   //........................Присваиваем обработанный выход к физическим выходам модуля...............................................................

   "AO V11.1" := "__MainBlock".Valve_Regul[1].iAnalogOutput;

   "AO V12.1" := "__MainBlock".Valve_Regul[2].iAnalogOutput;

   "AO V3 (NO)" := "__MainBlock".Valve_Regul[3].iAnalogOutput;

   //========================  Управление выходом пневмоострова для клапана регулировки============================
   //Управление клапанами через тройник от выходов запорных клапанов V11 и V12
   "__MainBlock".Valve_Regul[1].bAutoOpenClose := "V11_Запорный тепло";  //Сигнал на открытие регулировочного клапана паралельно с запорным клапаном
   "__MainBlock".Valve_Regul[2].bAutoOpenClose := "V12_Запор гликоль" ;   //Сигнал на открытие регулировочного клапана паралельно с запорным клапаном

   // Выход для управления клапаном V3
   "V3_Давления" := "__MainBlock".Valve_Regul[3].bOut_OpenClose;

   //=======================================//=======================================//=======================================//=======================================

   "__MainBlock".Valve_Regul[1].bManualOpenClose := "__MainBlock"."Valve_o/c"[11].bManualOpen;

   "__MainBlock".Valve_Regul[2].bManualOpenClose := "__MainBlock"."Valve_o/c"[12].bManualOpen;
END_FUNCTION

FUNCTION "Расчет ПЕ1" : Void   // FC9, LAD
{ S7_Optimized_Access := 'FALSE' }
VERSION : 0.1
   VAR_INPUT
      "ПЕ (ед)" : Int;
      "Выдержка (сек)" : Int;
      "Производит установки (л\ч)" : Int;
      "Производит заданная (л\ч)" : Int;
      "Уст.Темп (С)" : Real;   // Уставка температуры нагрева продукта
      "Выбор уставки для температуры (0 - ПЕ, 1 - Те)" : Bool;   // Для выбора от куда брать уставку температуры или вводим ПЕ и расчитываем ТЕ или просто вводим желаемую ПЕ
   END_VAR
   VAR_OUTPUT
      "Температура пастеризации" : Real;   // уставка для ПИД нагрева. Или расчитываем по ПЕ или по уставке желаемой ТЕ
      "Выдержка реальная_1" : Int;
      "Расчтеная ПЕ по Те" : Real;   // Расчет ПЕ по уставке Те для HMI
   END_VAR
   VAR_TEMP
      "1" : Real;
      "выдержка реальная" : Int;
      "2" : UInt;
      "3" : Real;
      "4" : Real;
      "5" : Real;
      "6" : Real;
      "Расчетная темп по ПЕ" : Real;   // Расчет температуры по уставке ПЕ
      "PE/10" : Int;
   END_VAR
   VAR CONSTANT
      "1.393" : Real := 1.393;
      "60" : Real := 60.0;
   END_VAR
BEGIN

REGION Network 1
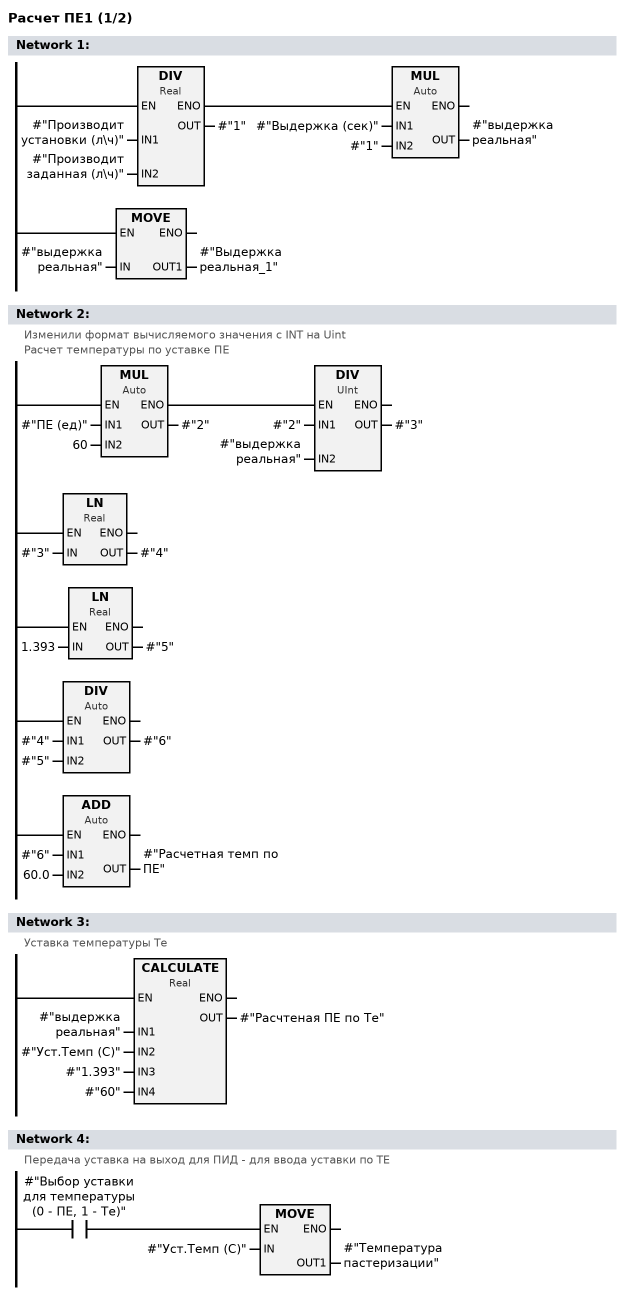
   RUNG wire#powerrail
      { S7_Templates := "SrcType := Real" } Div(in1 := #"Производит установки (л\ч)", in2 := #"Производит заданная (л\ч)", out => #"1")
      Mul(in1 := #"Выдержка (сек)", in2 := #"1", out => #"выдержка реальная")
   END_RUNG
   RUNG wire#powerrail
      Move(in := #"выдержка реальная", out1 => #"Выдержка реальная_1")
   END_RUNG
   // the same network as SCL:
   #"1" := #"Производит установки (л\ч)" / #"Производит заданная (л\ч)";
   #"выдержка реальная" := #"Выдержка (сек)" * #"1";
   #"Выдержка реальная_1" := #"выдержка реальная";
END_REGION

REGION Network 2
   // Изменили формат вычисляемого значения с INT на Uint
   // Расчет температуры по уставке ПЕ
   #"2" := #"ПЕ (ед)" * 60;
   #"3" := #"2" / #"выдержка реальная";
   #"4" := LN(#"3");
   #"5" := LN(1.393);
   #"6" := #"4" / #"5";
   #"Расчетная темп по ПЕ" := #"6" + 60.0;
END_REGION

REGION Network 3
   // Уставка температуры Те
   RUNG wire#powerrail
      { S7_Templates := "SrcType := Real"; S7_Expression := "IN1/IN4*(IN3**(IN2-IN4))" } Calculate(in1 := #"выдержка реальная", in2 := #"Уст.Темп (С)", in3 := #"1.393", in4 := #"60", out => #"Расчтеная ПЕ по Те")
   END_RUNG
   // the same network as SCL:
   #"Расчтеная ПЕ по Те" := #"выдержка реальная"/#"60"*(#"1.393"**(#"Уст.Темп (С)"-#"60"));
END_REGION

REGION Network 4
   // Передача уставка на выход для ПИД - для ввода уставки по ТЕ
   RUNG wire#powerrail
      Contact( #"Выбор уставки для температуры (0 - ПЕ, 1 - Те)" )
      Move(in := #"Уст.Темп (С)", out1 => #"Температура пастеризации")
   END_RUNG
   // the same network as SCL:
   IF #"Выбор уставки для температуры (0 - ПЕ, 1 - Те)" THEN
       #"Температура пастеризации" := #"Уст.Темп (С)";
   END_IF;
END_REGION

REGION Network 5
   // Передача уставка на выход для ПИД - для ввода уставки по ПЕ
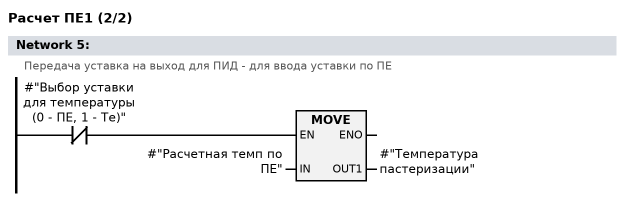
   RUNG wire#powerrail
      I_Contact( #"Выбор уставки для температуры (0 - ПЕ, 1 - Те)" )
      Move(in := #"Расчетная темп по ПЕ", out1 => #"Температура пастеризации")
   END_RUNG
   // the same network as SCL:
   IF NOT #"Выбор уставки для температуры (0 - ПЕ, 1 - Те)" THEN
       #"Температура пастеризации" := #"Расчетная темп по ПЕ";
   END_IF;
END_REGION
END_FUNCTION

FUNCTION "Все в Авто" : Void   // FC12, SCL
{ S7_Optimized_Access := 'TRUE' }
VERSION : 0.1
   VAR_TEMP
      fTrig_All_Auto : Bool;   // Фронт нажития кнопки все в авто
      i : Int;
   END_VAR
BEGIN

   //Отлавливаем фронт нажатия клавиши все в авто
   "R_trig_All_Auto"(In:="Клапана  в автомат",
                     Q=>#fTrig_All_Auto);

   //Сбрасываем все ручное в автоматический режим
   //
   IF #fTrig_All_Auto THEN

       //симуляция датчиков аналоговых
       //
       FOR #i := 1 TO 12 DO
           "__MainBlock".AI[#i].bSimEnable := FALSE;
       END_FOR;


       //Управление Valve o/c 
       FOR #i := 1 TO 20 DO
           "__MainBlock"."Valve_o/c"[#i].bManualMode := FALSE;
       END_FOR;

       //Управление Valve regul 
       FOR #i := 1 TO 3 DO
           "__MainBlock".Valve_Regul[#i].bManualMode := FALSE;
       END_FOR;


       //Управление Pumps
       FOR #i := 1 TO 6 DO
           "__MainBlock".Pump[#i].bManualMode := FALSE;
       END_FOR;



       //DI
       (*
       "DI".DI_0.bSimulation := FALSE;
       "DI".DI_1.bSimulation := FALSE;
       "DI".DI_2.bSimulation := FALSE;
       "DI".DI_3.bSimulation := FALSE;
       "DI".DI_4.bSimulation := FALSE;
       "DI".DI_5.bSimulation := FALSE;
       "DI".DI_6.bSimulation := FALSE;
       "DI".DI_7.bSimulation := FALSE;
       "DI".DI_8.bSimulation := FALSE;
       "DI".DI_9.bSimulation := FALSE;
       "DI".DI_10.bSimulation := FALSE;
       "DI".DI_11.bSimulation := FALSE;
       "DI".DI_12.bSimulation := FALSE;
       "DI".DI_13.bSimulation := FALSE;
       "DI".DI_14.bSimulation := FALSE;
       "DI".DI_15.bSimulation := FALSE;
       "DI".DI_16.bSimulation := FALSE;
       "DI".DI_17.bSimulation := FALSE;
       "DI".DI_18.bSimulation := FALSE;
       "DI".DI_19.bSimulation := FALSE;
       "DI".DI_20.bSimulation := FALSE;
       "DI".DI_21.bSimulation := FALSE;
       "DI".DI_22.bSimulation := FALSE;
       "DI".DI_23.bSimulation := FALSE;
       "DI".DI_24.bSimulation := FALSE;
       "DI".DI_25.bSimulation := FALSE;
       "DI".DI_26.bSimulation := FALSE;
       "DI".DI_27.bSimulation := FALSE;
       "DI".DI_28.bSimulation := FALSE;
       "DI".DI_29.bSimulation := FALSE;
      *)
   END_IF;
END_FUNCTION

FUNCTION "RestetAlarms" : Void   // FC13, SCL
{ S7_Optimized_Access := 'TRUE' }
VERSION : 0.1
   VAR_TEMP
      i : Int;
   END_VAR
BEGIN
   IF "bHMI_ResetAlarm" THEN

       //Сброс аварий насосов
       //
       FOR #i := 1 TO 6 DO
           "__MainBlock".Pump[#i].bResAlarm := TRUE;
       END_FOR;

       //Сброс аварий клапана
       //
       FOR #i := 1 TO 20 DO
           "__MainBlock"."Valve_o/c"[#i].bResetAlarm := TRUE;
       END_FOR;

   ELSE

       //Сброс аварий клапана
       FOR #i := 1 TO 20 DO
           "__MainBlock"."Valve_o/c"[#i].bResetAlarm := FALSE;
       END_FOR;

       //Сброс аварий насосов
       //
       FOR #i := 1 TO 6 DO
           "__MainBlock".Pump[#i].bResAlarm := FALSE;
       END_FOR;

   END_IF;
END_FUNCTION

ORGANIZATION_BLOCK "Main"   // OB1, LAD, ProgramCycle
TITLE = "Main Program Sweep (Cycle)"
{ S7_Optimized_Access := 'TRUE' }
AUTHOR : Алексей
VERSION : 0.1
   VAR_INPUT
      Initial_Call : Bool;   // Initial call of this OB
      Remanence : Bool;   // =True, if remanent data are available
   END_VAR
BEGIN

REGION Network 1: Расчет ПЕ
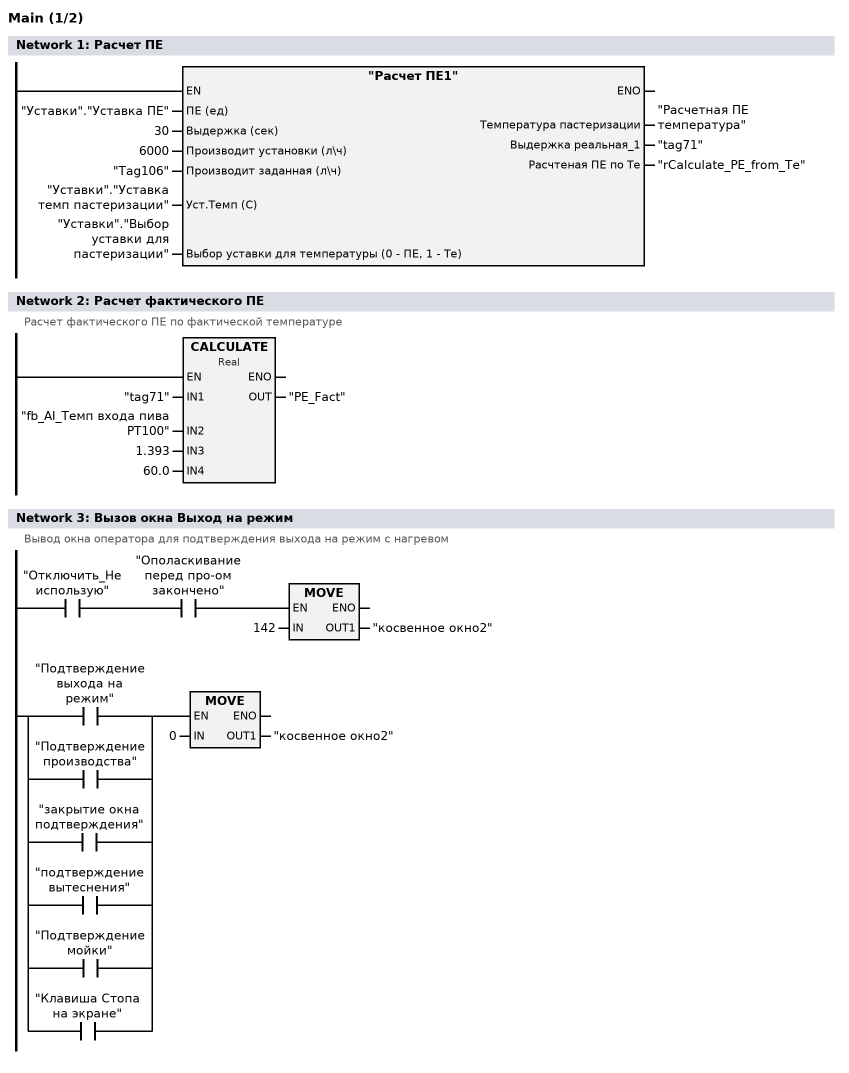
   RUNG wire#powerrail
      "Расчет ПЕ1"("ПЕ (ед)" := "Уставки"."Уставка ПЕ", "Выдержка (сек)" := 30, "Производит установки (л\ч)" := 6000, "Производит заданная (л\ч)" := "Tag106", "Уст.Темп (С)" := "Уставки"."Уставка темп пастеризации", "Выбор уставки для температуры (0 - ПЕ, 1 - Те)" := "Уставки"."Выбор уставки для пастеризации", "Температура пастеризации" => "Расчетная ПЕ температура", "Выдержка реальная_1" => "tag71", "Расчтеная ПЕ по Те" => "rCalculate_PE_from_Te")
   END_RUNG
   // the same network as SCL:
   "Расчет ПЕ1"("ПЕ (ед)" := "Уставки"."Уставка ПЕ",
                "Выдержка (сек)" := 30,
                "Производит установки (л\ч)" := 6000,
                "Производит заданная (л\ч)" := "Tag106",
                "Уст.Темп (С)" := "Уставки"."Уставка темп пастеризации",
                "Выбор уставки для температуры (0 - ПЕ, 1 - Те)" := "Уставки"."Выбор уставки для пастеризации",
                "Температура пастеризации" => "Расчетная ПЕ температура",
                "Выдержка реальная_1" => "tag71",
                "Расчтеная ПЕ по Те" => "rCalculate_PE_from_Te");
END_REGION

REGION Network 2: Расчет фактического ПЕ
   // Расчет фактического ПЕ по фактической температуре
   RUNG wire#powerrail
      { S7_Templates := "SrcType := Real"; S7_Expression := "IN1/IN4*(IN3**(IN2-IN4))" } Calculate(in1 := "tag71", in2 := "fb_AI_Темп входа пива PT100", in3 := 1.393, in4 := 60.0, out => "PE_Fact")
   END_RUNG
   // the same network as SCL:
   "PE_Fact" := "tag71"/60.0*(1.393**("fb_AI_Темп входа пива PT100"-60.0));
END_REGION

REGION Network 3: Вызов окна Выход на режим
   // Вывод окна оператора для подтверждения выхода на режим с нагревом
   RUNG wire#powerrail
      Contact( "Отключить_Не использую" )
      Contact( "Ополаскивание перед про-ом закончено" )
      Move(in := 142, out1 => "косвенное окно2")
   END_RUNG
   RUNG wire#powerrail
      Contact( "Подтверждение выхода на режим" )
      wire#w1
      Move(in := 0, out1 => "косвенное окно2")
   END_RUNG
   RUNG wire#powerrail
      Contact( "Подтверждение производства" )
   END_RUNG wire#w1
   RUNG wire#powerrail
      Contact( "закрытие окна подтверждения" )
   END_RUNG wire#w1
   RUNG wire#powerrail
      Contact( "подтверждение вытеснения" )
   END_RUNG wire#w1
   RUNG wire#powerrail
      Contact( "Подтверждение мойки" )
   END_RUNG wire#w1
   RUNG wire#powerrail
      Contact( "Клавиша Стопа на экране" )
   END_RUNG wire#w1
   // the same network as SCL:
   IF "Отключить_Не использую" AND "Ополаскивание перед про-ом закончено" THEN
       "косвенное окно2" := 142;
   END_IF;
   IF "Подтверждение выхода на режим" OR "Подтверждение производства" OR "закрытие окна подтверждения" OR "подтверждение вытеснения" OR "Подтверждение мойки" OR "Клавиша Стопа на экране" THEN
       "косвенное окно2" := 0;
   END_IF;
END_REGION

REGION Network 4: 11
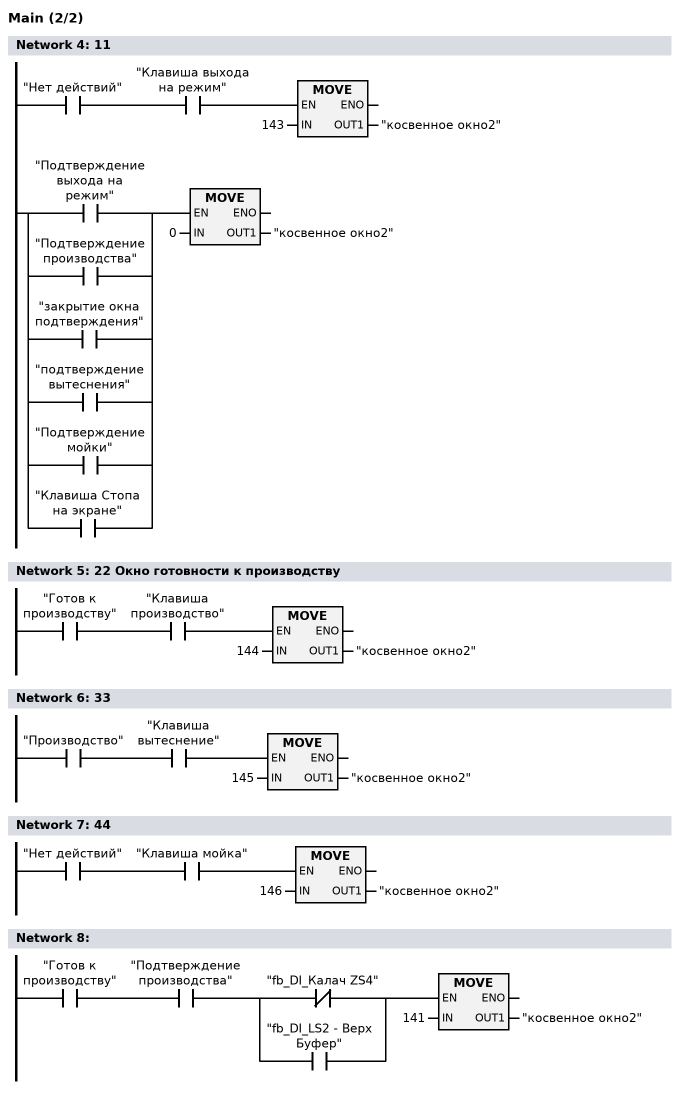
   RUNG wire#powerrail
      Contact( "Нет действий" )
      Contact( "Клавиша выхода на режим" )
      Move(in := 143, out1 => "косвенное окно2")
   END_RUNG
   RUNG wire#powerrail
      Contact( "Подтверждение выхода на режим" )
      wire#w1
      Move(in := 0, out1 => "косвенное окно2")
   END_RUNG
   RUNG wire#powerrail
      Contact( "Подтверждение производства" )
   END_RUNG wire#w1
   RUNG wire#powerrail
      Contact( "закрытие окна подтверждения" )
   END_RUNG wire#w1
   RUNG wire#powerrail
      Contact( "подтверждение вытеснения" )
   END_RUNG wire#w1
   RUNG wire#powerrail
      Contact( "Подтверждение мойки" )
   END_RUNG wire#w1
   RUNG wire#powerrail
      Contact( "Клавиша Стопа на экране" )
   END_RUNG wire#w1
   // the same network as SCL:
   IF "Нет действий" AND "Клавиша выхода на режим" THEN "косвенное окно2" := 143; END_IF;
   IF "Подтверждение выхода на режим" OR "Подтверждение производства" OR "закрытие окна подтверждения" OR "подтверждение вытеснения" OR "Подтверждение мойки" OR "Клавиша Стопа на экране" THEN
       "косвенное окно2" := 0;
   END_IF;
END_REGION

REGION Network 5: 22 Окно готовности к производству
   RUNG wire#powerrail
      Contact( "Готов к производству" )
      Contact( "Клавиша производство" )
      Move(in := 144, out1 => "косвенное окно2")
   END_RUNG
   // the same network as SCL:
   IF "Готов к производству" AND "Клавиша производство" THEN "косвенное окно2" := 144; END_IF;
END_REGION

REGION Network 6: 33
   RUNG wire#powerrail
      Contact( "Производство" )
      Contact( "Клавиша вытеснение" )
      Move(in := 145, out1 => "косвенное окно2")
   END_RUNG
   // the same network as SCL:
   IF "Производство" AND "Клавиша вытеснение" THEN "косвенное окно2" := 145; END_IF;
END_REGION

REGION Network 7: 44
   RUNG wire#powerrail
      Contact( "Нет действий" )
      Contact( "Клавиша мойка" )
      Move(in := 146, out1 => "косвенное окно2")
   END_RUNG
   // the same network as SCL:
   IF "Нет действий" AND "Клавиша мойка" THEN "косвенное окно2" := 146; END_IF;
END_REGION

REGION Network 8
   RUNG wire#powerrail
      Contact( "Готов к производству" )
      Contact( "Подтверждение производства" )
      wire#w1
      I_Contact( "fb_DI_Калач ZS4" )
      wire#w2
      Move(in := 141, out1 => "косвенное окно2")
   END_RUNG
   RUNG wire#w1
      Contact( "fb_DI_LS2 - Верх Буфер" )
   END_RUNG wire#w2
   // the same network as SCL:
   IF "Готов к производству" AND "Подтверждение производства" AND (NOT "fb_DI_Калач ZS4" OR "fb_DI_LS2 - Верх Буфер") THEN
       "косвенное окно2" := 141;
   END_IF;
END_REGION
END_ORGANIZATION_BLOCK

ORGANIZATION_BLOCK "Масштабирование"   // OB123, LAD, ProgramCycle
TITLE = "Main Program Sweep (Cycle)"
{ S7_Optimized_Access := 'TRUE' }
VERSION : 0.1
   VAR_INPUT
      Initial_Call : Bool;   // Initial call of this OB
      Remanence : Bool;   // =True, if remanent data are available
   END_VAR
   VAR_TEMP
      a1 : Real;
      a2 : Real;
      a3 : Real;
      a4 : Real;
      a5 : Real;
      a6 : Real;
      a7 : Real;
      a8 : Real;
      a9 : Real;
   END_VAR
BEGIN

REGION Network 1: Температура выхода продукта
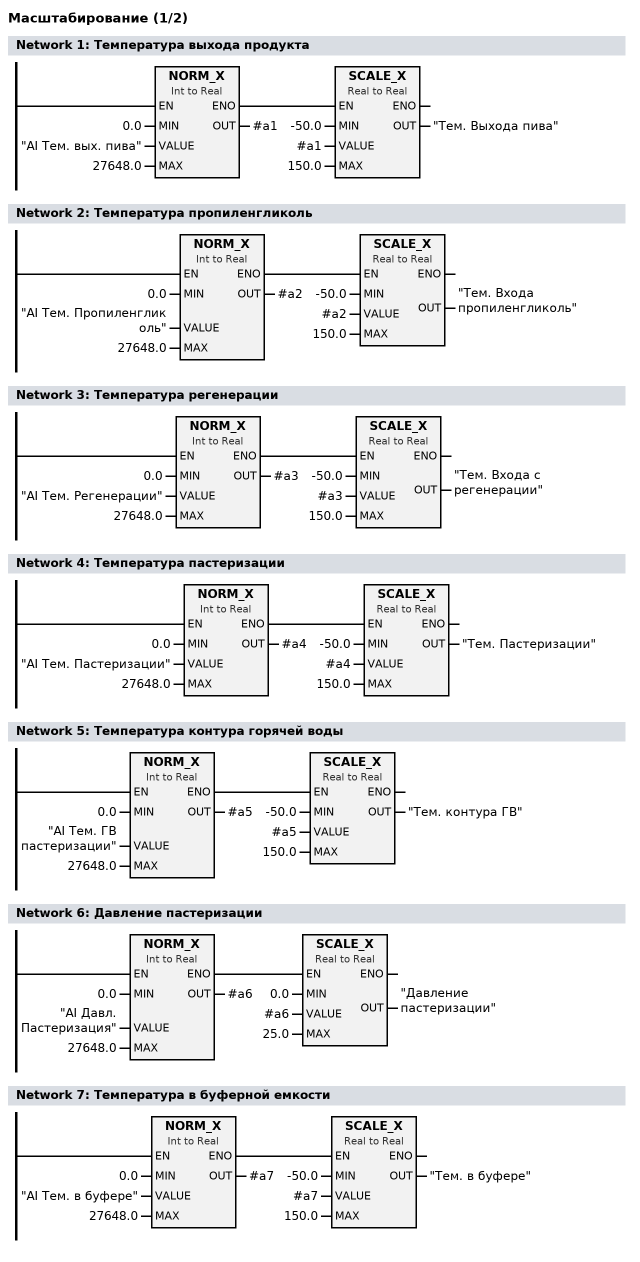
   RUNG wire#powerrail
      { S7_Templates := "[SrcType := Int, DestType := Real]" } Normalize(min := 0.0, value := "AI Тем. вых. пива", max := 27648.0, out => #a1)
      { S7_Templates := "[SrcType := Real, DestType := Real]" } Scale(min := -50.0, value := #a1, max := 150.0, out => "Тем. Выхода пива")
   END_RUNG
   // the same network as SCL:
   #a1 := NORM_X(MIN := 0.0, VALUE := "AI Тем. вых. пива", MAX := 27648.0);
   "Тем. Выхода пива" := SCALE_X(MIN := -50.0, VALUE := #a1, MAX := 150.0);
END_REGION

REGION Network 2: Температура пропиленгликоль
   RUNG wire#powerrail
      { S7_Templates := "[SrcType := Int, DestType := Real]" } Normalize(min := 0.0, value := "AI Тем. Пропиленгликоль", max := 27648.0, out => #a2)
      { S7_Templates := "[SrcType := Real, DestType := Real]" } Scale(min := -50.0, value := #a2, max := 150.0, out => "Тем. Входа пропиленгликоль")
   END_RUNG
   // the same network as SCL:
   #a2 := NORM_X(MIN := 0.0, VALUE := "AI Тем. Пропиленгликоль", MAX := 27648.0);
   "Тем. Входа пропиленгликоль" := SCALE_X(MIN := -50.0, VALUE := #a2, MAX := 150.0);
END_REGION

REGION Network 3: Температура регенерации
   RUNG wire#powerrail
      { S7_Templates := "[SrcType := Int, DestType := Real]" } Normalize(min := 0.0, value := "AI Тем. Регенерации", max := 27648.0, out => #a3)
      { S7_Templates := "[SrcType := Real, DestType := Real]" } Scale(min := -50.0, value := #a3, max := 150.0, out => "Тем. Входа с регенерации")
   END_RUNG
   // the same network as SCL:
   #a3 := NORM_X(MIN := 0.0, VALUE := "AI Тем. Регенерации", MAX := 27648.0);
   "Тем. Входа с регенерации" := SCALE_X(MIN := -50.0, VALUE := #a3, MAX := 150.0);
END_REGION

REGION Network 4: Температура пастеризации
   RUNG wire#powerrail
      { S7_Templates := "[SrcType := Int, DestType := Real]" } Normalize(min := 0.0, value := "AI Тем. Пастеризации", max := 27648.0, out => #a4)
      { S7_Templates := "[SrcType := Real, DestType := Real]" } Scale(min := -50.0, value := #a4, max := 150.0, out => "Тем. Пастеризации")
   END_RUNG
   // the same network as SCL:
   #a4 := NORM_X(MIN := 0.0, VALUE := "AI Тем. Пастеризации", MAX := 27648.0);
   "Тем. Пастеризации" := SCALE_X(MIN := -50.0, VALUE := #a4, MAX := 150.0);
END_REGION

REGION Network 5: Температура контура горячей воды
   RUNG wire#powerrail
      { S7_Templates := "[SrcType := Int, DestType := Real]" } Normalize(min := 0.0, value := "AI Тем. ГВ пастеризации", max := 27648.0, out => #a5)
      { S7_Templates := "[SrcType := Real, DestType := Real]" } Scale(min := -50.0, value := #a5, max := 150.0, out => "Тем. контура ГВ")
   END_RUNG
   // the same network as SCL:
   #a5 := NORM_X(MIN := 0.0, VALUE := "AI Тем. ГВ пастеризации", MAX := 27648.0);
   "Тем. контура ГВ" := SCALE_X(MIN := -50.0, VALUE := #a5, MAX := 150.0);
END_REGION

REGION Network 6: Давление пастеризации
   RUNG wire#powerrail
      { S7_Templates := "[SrcType := Int, DestType := Real]" } Normalize(min := 0.0, value := "AI Давл. Пастеризация", max := 27648.0, out => #a6)
      { S7_Templates := "[SrcType := Real, DestType := Real]" } Scale(min := 0.0, value := #a6, max := 25.0, out => "Давление пастеризации")
   END_RUNG
   // the same network as SCL:
   #a6 := NORM_X(MIN := 0.0, VALUE := "AI Давл. Пастеризация", MAX := 27648.0);
   "Давление пастеризации" := SCALE_X(MIN := 0.0, VALUE := #a6, MAX := 25.0);
END_REGION

REGION Network 7: Температура в буферной емкости
   RUNG wire#powerrail
      { S7_Templates := "[SrcType := Int, DestType := Real]" } Normalize(min := 0.0, value := "AI Тем. в буфере", max := 27648.0, out => #a7)
      { S7_Templates := "[SrcType := Real, DestType := Real]" } Scale(min := -50.0, value := #a7, max := 150.0, out => "Тем. в буфере")
   END_RUNG
   // the same network as SCL:
   #a7 := NORM_X(MIN := 0.0, VALUE := "AI Тем. в буфере", MAX := 27648.0);
   "Тем. в буфере" := SCALE_X(MIN := -50.0, VALUE := #a7, MAX := 150.0);
END_REGION

REGION Network 8: Датчик давления на розливе
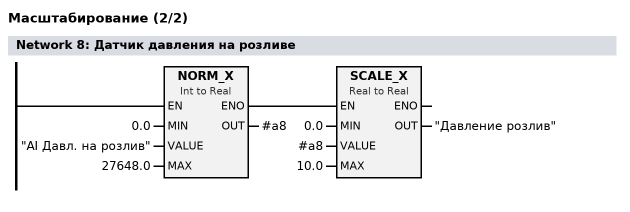
   RUNG wire#powerrail
      { S7_Templates := "[SrcType := Int, DestType := Real]" } Normalize(min := 0.0, value := "AI Давл. на розлив", max := 27648.0, out => #a8)
      { S7_Templates := "[SrcType := Real, DestType := Real]" } Scale(min := 0.0, value := #a8, max := 10.0, out => "Давление розлив")
   END_RUNG
   // the same network as SCL:
   #a8 := NORM_X(MIN := 0.0, VALUE := "AI Давл. на розлив", MAX := 27648.0);
   "Давление розлив" := SCALE_X(MIN := 0.0, VALUE := #a8, MAX := 10.0);
END_REGION
END_ORGANIZATION_BLOCK

ORGANIZATION_BLOCK "Реж_Выход на режим кольцо"   // OB124, LAD, ProgramCycle
TITLE = "Main Program Sweep (Cycle)"
{ S7_Optimized_Access := 'TRUE' }
VERSION : 0.1
   VAR_INPUT
      Initial_Call : Bool;   // Initial call of this OB
      Remanence : Bool;   // =True, if remanent data are available
   END_VAR
   VAR_TEMP   // added for the SCL form of the ladder/FBD networks
      _w1 : Bool;
   END_VAR
BEGIN

REGION Network 1: Заполнение Водой
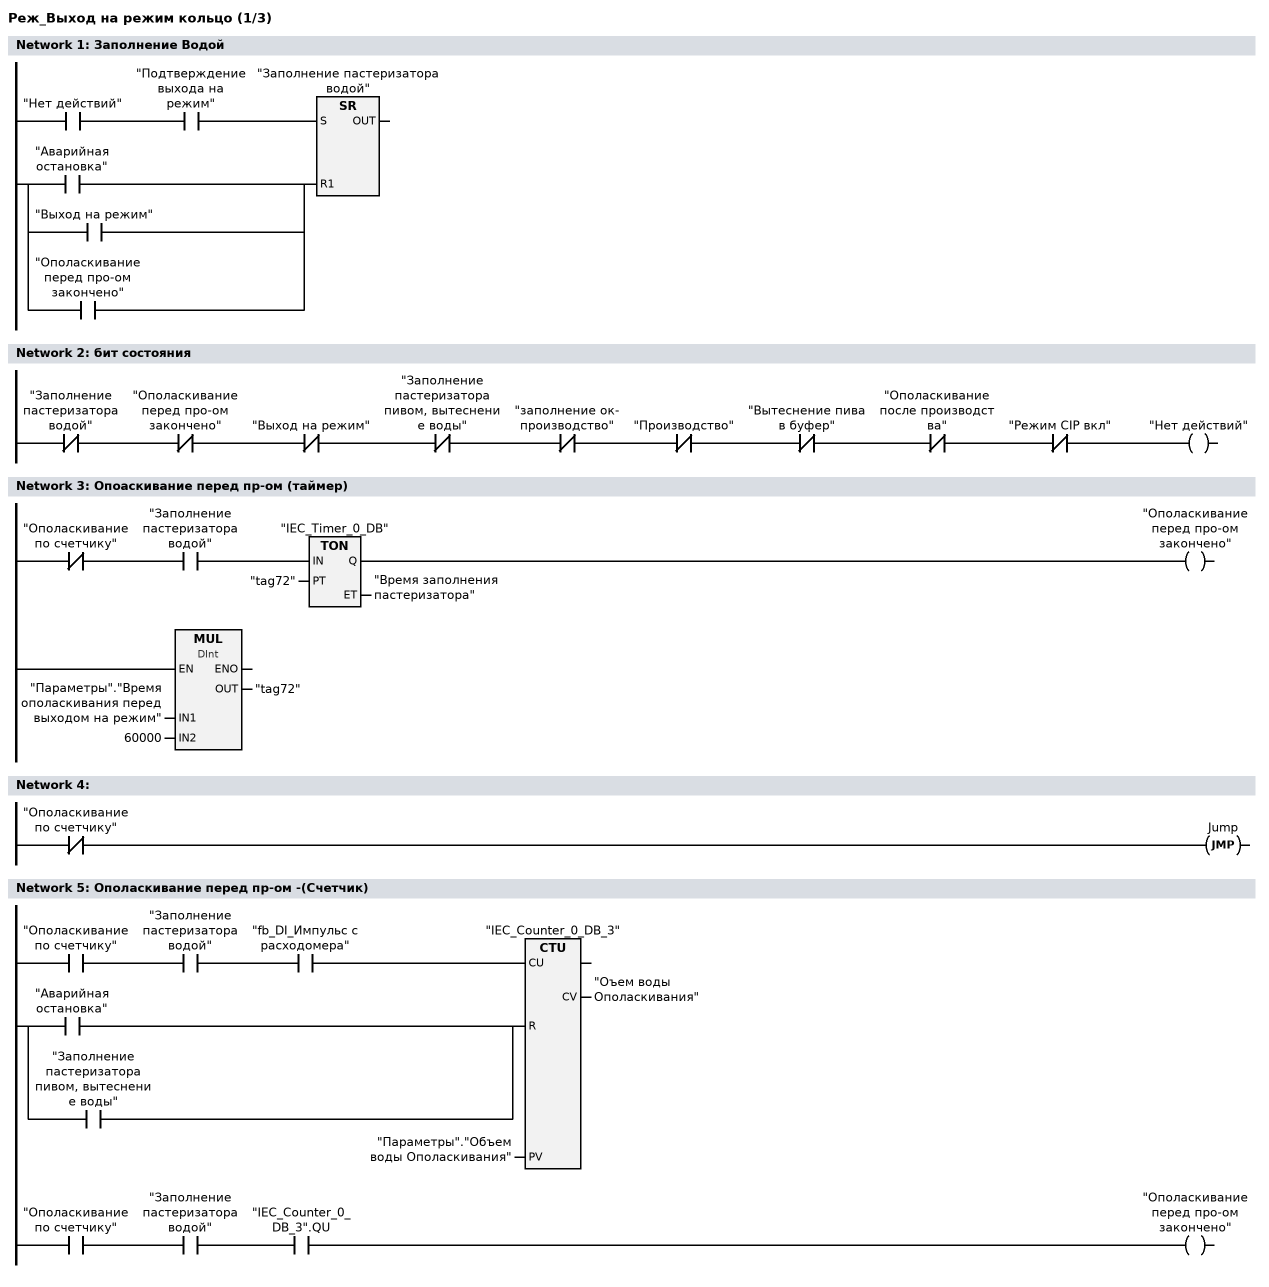
   RUNG wire#powerrail
      Contact( "Нет действий" )
      Contact( "Подтверждение выхода на режим" )
      S_SR(operand := "Заполнение пастеризатора водой", r1 := wire#w1)
   END_RUNG
   RUNG wire#powerrail
      Contact( "Аварийная остановка" )
   END_RUNG wire#w1
   RUNG wire#powerrail
      Contact( "Выход на режим" )
   END_RUNG wire#w1
   RUNG wire#powerrail
      Contact( "Ополаскивание перед про-ом закончено" )
   END_RUNG wire#w1
   // the same network as SCL:
   IF "Нет действий" AND "Подтверждение выхода на режим" THEN
       "Заполнение пастеризатора водой" := TRUE;   // SR flip-flop
   END_IF;
   IF "Аварийная остановка" OR "Выход на режим" OR "Ополаскивание перед про-ом закончено" THEN
       "Заполнение пастеризатора водой" := FALSE;
   END_IF;
END_REGION

REGION Network 2: бит состояния
   RUNG wire#powerrail
      I_Contact( "Заполнение пастеризатора водой" )
      I_Contact( "Ополаскивание перед про-ом закончено" )
      I_Contact( "Выход на режим" )
      I_Contact( "Заполнение пастеризатора пивом, вытеснение воды" )
      I_Contact( "заполнение ок- производство" )
      I_Contact( "Производство" )
      I_Contact( "Вытеснение пива в буфер" )
      I_Contact( "Ополаскивание после производства" )
      I_Contact( "Режим СIP вкл" )
      Coil( "Нет действий" )
   END_RUNG
   // the same network as SCL:
   "Нет действий" := NOT "Заполнение пастеризатора водой" AND NOT "Ополаскивание перед про-ом закончено" AND NOT "Выход на режим" AND NOT "Заполнение пастеризатора пивом, вытеснение воды" AND NOT "заполнение ок- производство" AND NOT "Производство" AND NOT "Вытеснение пива в буфер" AND NOT "Ополаскивание после производства" AND NOT "Режим СIP вкл";
END_REGION

REGION Network 3: Опоаскивание перед пр-ом (таймер)
   "IEC_Timer_0_DB".TON(IN := NOT "Ополаскивание по счетчику" AND "Заполнение пастеризатора водой",
                        PT := "tag72",
                        ET => "Время заполнения пастеризатора");
   "Ополаскивание перед про-ом закончено" := "IEC_Timer_0_DB".Q;
   "tag72" := "Параметры"."Время ополаскивания перед выходом на режим" * 60000;
END_REGION

REGION Network 4
   RUNG wire#powerrail
      I_Contact( "Ополаскивание по счетчику" )
      JumpCoil( Jump )
   END_RUNG
   // the same network as SCL:
   IF NOT "Ополаскивание по счетчику" THEN GOTO Jump; END_IF;
END_REGION

REGION Network 5: Ополаскивание перед пр-ом -(Счетчик)
   "IEC_Counter_0_DB_3".CTU(CU := "Ополаскивание по счетчику" AND "Заполнение пастеризатора водой" AND "fb_DI_Импульс с расходомера",
                           R := "Аварийная остановка" OR "Заполнение пастеризатора пивом, вытеснение воды",
                           PV := "Параметры"."Объем воды Ополаскивания",
                           CV => "Оъем воды Ополаскивания");
   "Ополаскивание перед про-ом закончено" := "Ополаскивание по счетчику" AND "Заполнение пастеризатора водой" AND "IEC_Counter_0_DB_3".QU;
END_REGION

REGION Network 6: Выход на режим
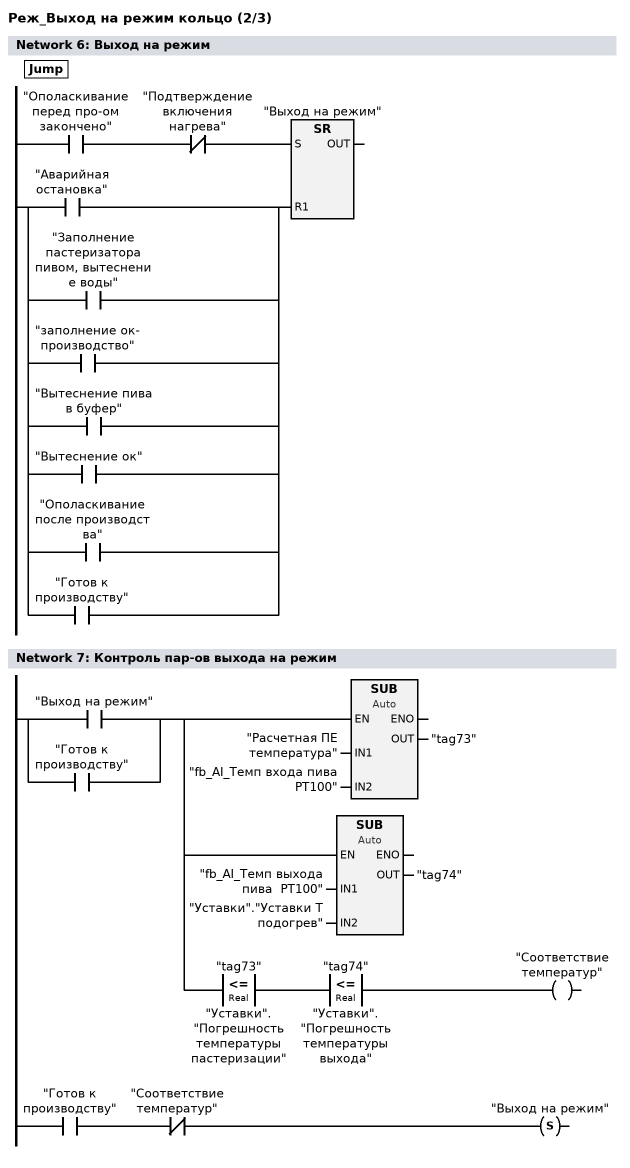
   Label( Jump )
   RUNG wire#powerrail
      Contact( "Ополаскивание перед про-ом закончено" )
      I_Contact( "Подтверждение включения нагрева" )
      S_SR(operand := "Выход на режим", r1 := wire#w1)
   END_RUNG
   RUNG wire#powerrail
      Contact( "Аварийная остановка" )
   END_RUNG wire#w1
   RUNG wire#powerrail
      Contact( "Заполнение пастеризатора пивом, вытеснение воды" )
   END_RUNG wire#w1
   RUNG wire#powerrail
      Contact( "заполнение ок- производство" )
   END_RUNG wire#w1
   RUNG wire#powerrail
      Contact( "Вытеснение пива в буфер" )
   END_RUNG wire#w1
   RUNG wire#powerrail
      Contact( "Вытеснение ок" )
   END_RUNG wire#w1
   RUNG wire#powerrail
      Contact( "Ополаскивание после производства" )
   END_RUNG wire#w1
   RUNG wire#powerrail
      Contact( "Готов к производству" )
   END_RUNG wire#w1
   // the same network as SCL:
   Jump:
   IF "Ополаскивание перед про-ом закончено" AND NOT "Подтверждение включения нагрева" THEN
       "Выход на режим" := TRUE;   // SR flip-flop
   END_IF;
   IF "Аварийная остановка" OR "Заполнение пастеризатора пивом, вытеснение воды" OR "заполнение ок- производство" OR "Вытеснение пива в буфер" OR "Вытеснение ок" OR "Ополаскивание после производства" OR "Готов к производству" THEN
       "Выход на режим" := FALSE;
   END_IF;
END_REGION

REGION Network 7: Контроль пар-ов выхода на режим
   RUNG wire#powerrail
      Contact( "Выход на режим" )
      wire#w1
      Sub(in1 := "Расчетная ПЕ температура", in2 := "fb_AI_Темп входа пива PT100", out => "tag73")
   END_RUNG
   RUNG wire#powerrail
      Contact( "Готов к производству" )
   END_RUNG wire#w1
   RUNG wire#w1
      Sub(in1 := "fb_AI_Темп выхода пива  PT100", in2 := "Уставки"."Уставки Т подогрев", out => "tag74")
   END_RUNG
   RUNG wire#w1
      { S7_Templates := "SrcType := Real" } LE_Contact(in1 := "tag73", in2 := "Уставки"."Погрешность температуры пастеризации")
      { S7_Templates := "SrcType := Real" } LE_Contact(in1 := "tag74", in2 := "Уставки"."Погрешность температуры выхода")
      Coil( "Соответствие температур" )
   END_RUNG
   RUNG wire#powerrail
      Contact( "Готов к производству" )
      I_Contact( "Соответствие температур" )
      S_Coil( "Выход на режим" )
   END_RUNG
   // the same network as SCL:
   #_w1 := "Выход на режим" OR "Готов к производству";
   IF #_w1 THEN
       "tag73" := "Расчетная ПЕ температура" - "fb_AI_Темп входа пива PT100";
       "tag74" := "fb_AI_Темп выхода пива  PT100" - "Уставки"."Уставки Т подогрев";
   END_IF;
   "Соответствие температур" := #_w1 AND ("tag73" <= "Уставки"."Погрешность температуры пастеризации") AND ("tag74" <= "Уставки"."Погрешность температуры выхода");
   IF "Готов к производству" AND NOT "Соответствие температур" THEN "Выход на режим" := TRUE; END_IF;
END_REGION

REGION Network 8: Переход в Готов к производству
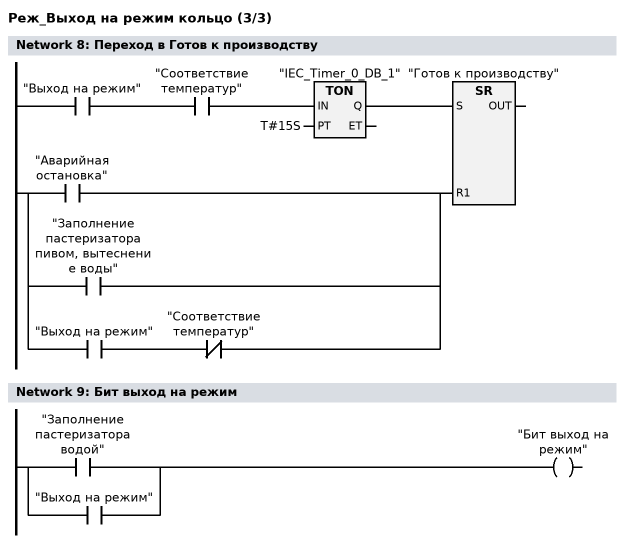
   "IEC_Timer_0_DB_1".TON(IN := "Выход на режим" AND "Соответствие температур", PT := T#15S);
   IF "IEC_Timer_0_DB_1".Q THEN
       "Готов к производству" := TRUE;   // SR flip-flop
   END_IF;
   IF "Аварийная остановка" OR "Заполнение пастеризатора пивом, вытеснение воды" OR ("Выход на режим" AND NOT "Соответствие температур") THEN
       "Готов к производству" := FALSE;
   END_IF;
END_REGION

REGION Network 9: Бит выход на режим
   RUNG wire#powerrail
      Contact( "Заполнение пастеризатора водой" )
      wire#w1
      Coil( "Бит выход на режим" )
   END_RUNG
   RUNG wire#powerrail
      Contact( "Выход на режим" )
   END_RUNG wire#w1
   // the same network as SCL:
   "Бит выход на режим" := "Заполнение пастеризатора водой" OR "Выход на режим";
END_REGION
END_ORGANIZATION_BLOCK

ORGANIZATION_BLOCK "Выхода"   // OB125, LAD, ProgramCycle
TITLE = "Main Program Sweep (Cycle)"
{ S7_Optimized_Access := 'TRUE' }
VERSION : 0.1
   VAR_INPUT
      Initial_Call : Bool;   // Initial call of this OB
      Remanence : Bool;   // =True, if remanent data are available
   END_VAR
BEGIN

REGION Network 1: Ручной режим
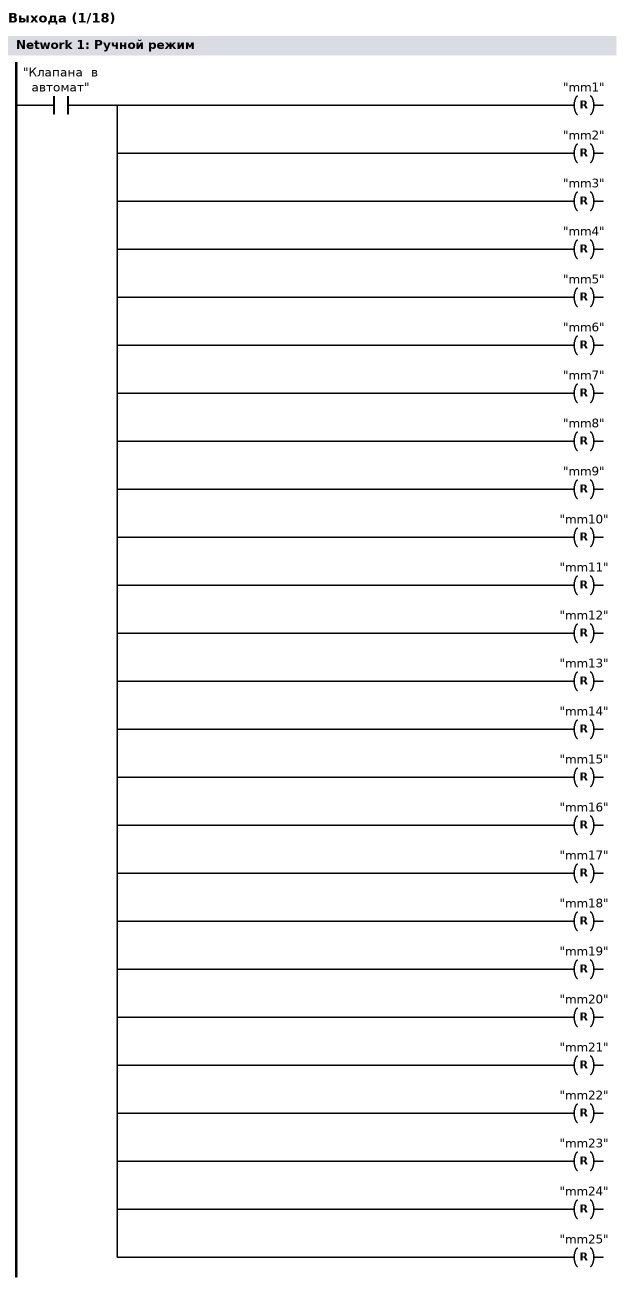
   RUNG wire#powerrail
      Contact( "Клапана  в автомат" )
      wire#w1
      R_Coil( "mm1" )
   END_RUNG
   RUNG wire#w1
      R_Coil( "mm2" )
   END_RUNG
   RUNG wire#w1
      R_Coil( "mm3" )
   END_RUNG
   RUNG wire#w1
      R_Coil( "mm4" )
   END_RUNG
   RUNG wire#w1
      R_Coil( "mm5" )
   END_RUNG
   RUNG wire#w1
      R_Coil( "mm6" )
   END_RUNG
   RUNG wire#w1
      R_Coil( "mm7" )
   END_RUNG
   RUNG wire#w1
      R_Coil( "mm8" )
   END_RUNG
   RUNG wire#w1
      R_Coil( "mm9" )
   END_RUNG
   RUNG wire#w1
      R_Coil( "mm10" )
   END_RUNG
   RUNG wire#w1
      R_Coil( "mm11" )
   END_RUNG
   RUNG wire#w1
      R_Coil( "mm12" )
   END_RUNG
   RUNG wire#w1
      R_Coil( "mm13" )
   END_RUNG
   RUNG wire#w1
      R_Coil( "mm14" )
   END_RUNG
   RUNG wire#w1
      R_Coil( "mm15" )
   END_RUNG
   RUNG wire#w1
      R_Coil( "mm16" )
   END_RUNG
   RUNG wire#w1
      R_Coil( "mm17" )
   END_RUNG
   RUNG wire#w1
      R_Coil( "mm18" )
   END_RUNG
   RUNG wire#w1
      R_Coil( "mm19" )
   END_RUNG
   RUNG wire#w1
      R_Coil( "mm20" )
   END_RUNG
   RUNG wire#w1
      R_Coil( "mm21" )
   END_RUNG
   RUNG wire#w1
      R_Coil( "mm22" )
   END_RUNG
   RUNG wire#w1
      R_Coil( "mm23" )
   END_RUNG
   RUNG wire#w1
      R_Coil( "mm24" )
   END_RUNG
   RUNG wire#w1
      R_Coil( "mm25" )
   END_RUNG
   // the same network as SCL:
   IF "Клапана  в автомат" THEN
       "mm1" := FALSE;
       "mm2" := FALSE;
       "mm3" := FALSE;
       "mm4" := FALSE;
       "mm5" := FALSE;
       "mm6" := FALSE;
       "mm7" := FALSE;
       "mm8" := FALSE;
       "mm9" := FALSE;
       "mm10" := FALSE;
       "mm11" := FALSE;
       "mm12" := FALSE;
       "mm13" := FALSE;
       "mm14" := FALSE;
       "mm15" := FALSE;
       "mm16" := FALSE;
       "mm17" := FALSE;
       "mm18" := FALSE;
       "mm19" := FALSE;
       "mm20" := FALSE;
       "mm21" := FALSE;
       "mm22" := FALSE;
       "mm23" := FALSE;
       "mm24" := FALSE;
       "mm25" := FALSE;
   END_IF;
END_REGION

REGION Network 2: Зеленый
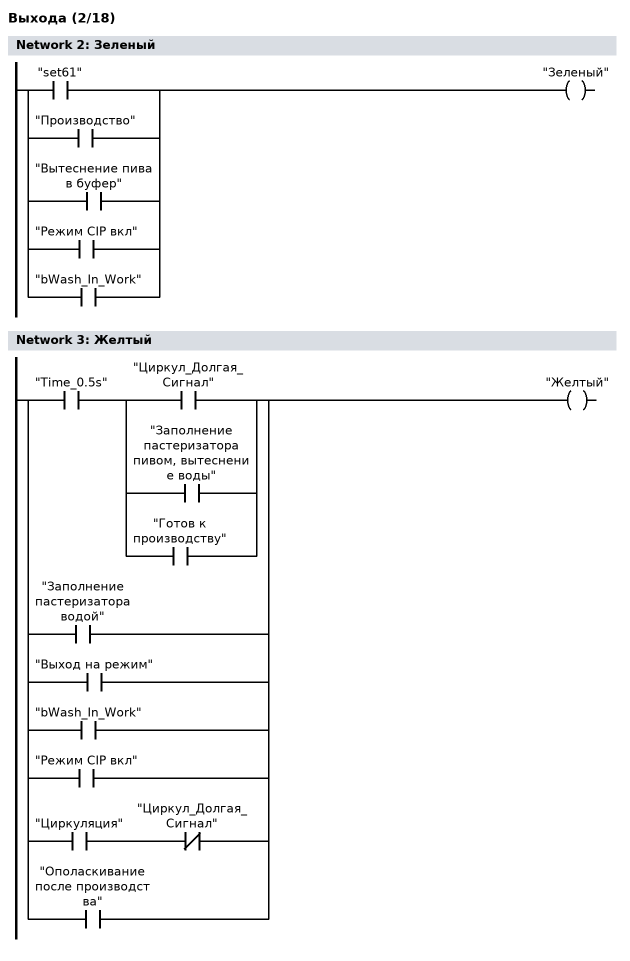
   RUNG wire#powerrail
      Contact( "set61" )
      wire#w1
      Coil( "Зеленый" )
   END_RUNG
   RUNG wire#powerrail
      Contact( "Производство" )
   END_RUNG wire#w1
   RUNG wire#powerrail
      Contact( "Вытеснение пива в буфер" )
   END_RUNG wire#w1
   RUNG wire#powerrail
      Contact( "Режим СIP вкл" )
   END_RUNG wire#w1
   RUNG wire#powerrail
      Contact( "bWash_In_Work" )
   END_RUNG wire#w1
   // the same network as SCL:
   "Зеленый" := "set61" OR "Производство" OR "Вытеснение пива в буфер" OR "Режим СIP вкл" OR "bWash_In_Work";
END_REGION

REGION Network 3: Желтый
   RUNG wire#powerrail
      Contact( "Time_0.5s" )
      wire#w1
      Contact( "Циркул_Долгая_Сигнал" )
      wire#w2
      Coil( "Желтый" )
   END_RUNG
   RUNG wire#w1
      Contact( "Заполнение пастеризатора пивом, вытеснение воды" )
   END_RUNG wire#w2
   RUNG wire#w1
      Contact( "Готов к производству" )
   END_RUNG wire#w2
   RUNG wire#powerrail
      Contact( "Заполнение пастеризатора водой" )
   END_RUNG wire#w2
   RUNG wire#powerrail
      Contact( "Выход на режим" )
   END_RUNG wire#w2
   RUNG wire#powerrail
      Contact( "bWash_In_Work" )
   END_RUNG wire#w2
   RUNG wire#powerrail
      Contact( "Режим СIP вкл" )
   END_RUNG wire#w2
   RUNG wire#powerrail
      Contact( "Циркуляция" )
      I_Contact( "Циркул_Долгая_Сигнал" )
   END_RUNG wire#w2
   RUNG wire#powerrail
      Contact( "Ополаскивание после производства" )
   END_RUNG wire#w2
   // the same network as SCL:
   "Желтый" := ("Time_0.5s" AND ("Циркул_Долгая_Сигнал" OR "Заполнение пастеризатора пивом, вытеснение воды" OR "Готов к производству")) OR "Заполнение пастеризатора водой" OR "Выход на режим" OR "bWash_In_Work" OR "Режим СIP вкл" OR ("Циркуляция" AND NOT "Циркул_Долгая_Сигнал") OR "Ополаскивание после производства";
END_REGION

REGION Network 4: Красный
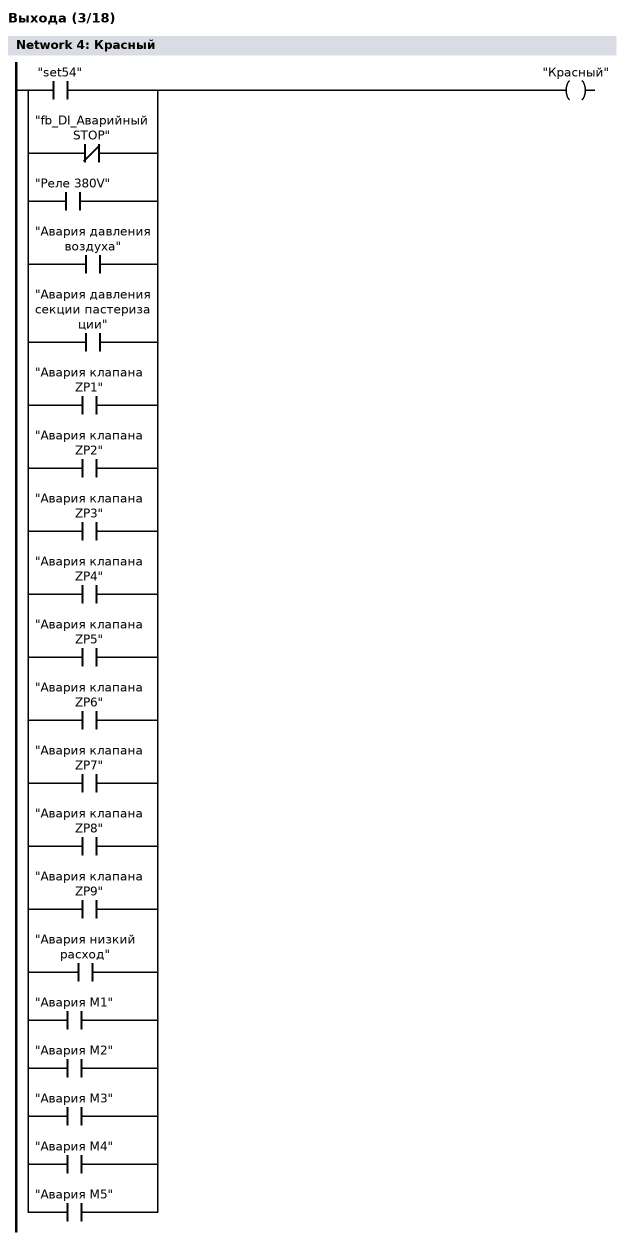
   RUNG wire#powerrail
      Contact( "set54" )
      wire#w1
      Coil( "Красный" )
   END_RUNG
   RUNG wire#powerrail
      I_Contact( "fb_DI_Аварийный STOP" )
   END_RUNG wire#w1
   RUNG wire#powerrail
      Contact( "Реле 380V" )
   END_RUNG wire#w1
   RUNG wire#powerrail
      Contact( "Авария давления воздуха" )
   END_RUNG wire#w1
   RUNG wire#powerrail
      Contact( "Авария давления секции пастеризации" )
   END_RUNG wire#w1
   RUNG wire#powerrail
      Contact( "Авария клапана ZP1" )
   END_RUNG wire#w1
   RUNG wire#powerrail
      Contact( "Авария клапана ZP2" )
   END_RUNG wire#w1
   RUNG wire#powerrail
      Contact( "Авария клапана ZP3" )
   END_RUNG wire#w1
   RUNG wire#powerrail
      Contact( "Авария клапана ZP4" )
   END_RUNG wire#w1
   RUNG wire#powerrail
      Contact( "Авария клапана ZP5" )
   END_RUNG wire#w1
   RUNG wire#powerrail
      Contact( "Авария клапана ZP6" )
   END_RUNG wire#w1
   RUNG wire#powerrail
      Contact( "Авария клапана ZP7" )
   END_RUNG wire#w1
   RUNG wire#powerrail
      Contact( "Авария клапана ZP8" )
   END_RUNG wire#w1
   RUNG wire#powerrail
      Contact( "Авария клапана ZP9" )
   END_RUNG wire#w1
   RUNG wire#powerrail
      Contact( "Авария низкий расход" )
   END_RUNG wire#w1
   RUNG wire#powerrail
      Contact( "Авария M1" )
   END_RUNG wire#w1
   RUNG wire#powerrail
      Contact( "Авария М2" )
   END_RUNG wire#w1
   RUNG wire#powerrail
      Contact( "Авария М3" )
   END_RUNG wire#w1
   RUNG wire#powerrail
      Contact( "Авария М4" )
   END_RUNG wire#w1
   RUNG wire#powerrail
      Contact( "Авария М5" )
   END_RUNG wire#w1
   // the same network as SCL:
   "Красный" := "set54" OR NOT "fb_DI_Аварийный STOP" OR "Реле 380V" OR "Авария давления воздуха" OR "Авария давления секции пастеризации" OR "Авария клапана ZP1" OR "Авария клапана ZP2" OR "Авария клапана ZP3" OR "Авария клапана ZP4" OR "Авария клапана ZP5" OR "Авария клапана ZP6" OR "Авария клапана ZP7" OR "Авария клапана ZP8" OR "Авария клапана ZP9" OR "Авария низкий расход" OR "Авария M1" OR "Авария М2" OR "Авария М3" OR "Авария М4" OR "Авария М5";
END_REGION

REGION Network 5: Сирена
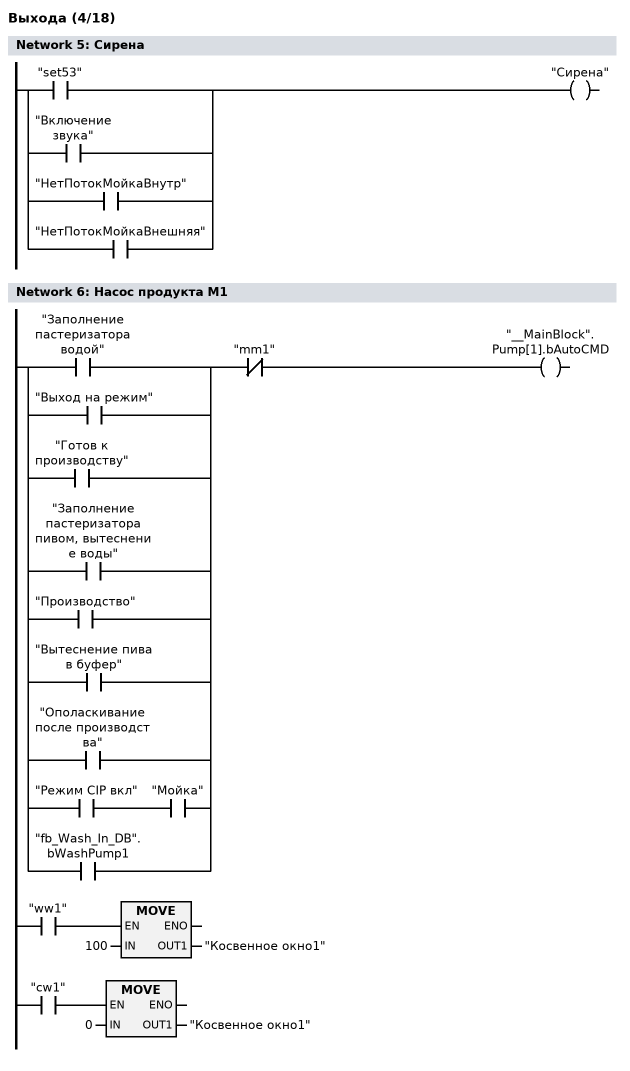
   RUNG wire#powerrail
      Contact( "set53" )
      wire#w1
      Coil( "Сирена" )
   END_RUNG
   RUNG wire#powerrail
      Contact( "Включение звука" )
   END_RUNG wire#w1
   RUNG wire#powerrail
      Contact( "НетПотокМойкаВнутр" )
   END_RUNG wire#w1
   RUNG wire#powerrail
      Contact( "НетПотокМойкаВнешняя" )
   END_RUNG wire#w1
   // the same network as SCL:
   "Сирена" := "set53" OR "Включение звука" OR "НетПотокМойкаВнутр" OR "НетПотокМойкаВнешняя";
END_REGION

REGION Network 6: Насос продукта M1
   RUNG wire#powerrail
      Contact( "Заполнение пастеризатора водой" )
      wire#w1
      I_Contact( "mm1" )
      Coil( "__MainBlock".Pump[1].bAutoCMD )
   END_RUNG
   RUNG wire#powerrail
      Contact( "Выход на режим" )
   END_RUNG wire#w1
   RUNG wire#powerrail
      Contact( "Готов к производству" )
   END_RUNG wire#w1
   RUNG wire#powerrail
      Contact( "Заполнение пастеризатора пивом, вытеснение воды" )
   END_RUNG wire#w1
   RUNG wire#powerrail
      Contact( "Производство" )
   END_RUNG wire#w1
   RUNG wire#powerrail
      Contact( "Вытеснение пива в буфер" )
   END_RUNG wire#w1
   RUNG wire#powerrail
      Contact( "Ополаскивание после производства" )
   END_RUNG wire#w1
   RUNG wire#powerrail
      Contact( "Режим СIP вкл" )
      Contact( "Мойка" )
   END_RUNG wire#w1
   RUNG wire#powerrail
      Contact( "fb_Wash_In_DB".bWashPump1 )
   END_RUNG wire#w1
   RUNG wire#powerrail
      Contact( "ww1" )
      Move(in := 100, out1 => "Косвенное окно1")
   END_RUNG
   RUNG wire#powerrail
      Contact( "cw1" )
      Move(in := 0, out1 => "Косвенное окно1")
   END_RUNG
   // the same network as SCL:
   "__MainBlock".Pump[1].bAutoCMD := ("Заполнение пастеризатора водой" OR "Выход на режим" OR "Готов к производству" OR "Заполнение пастеризатора пивом, вытеснение воды" OR "Производство" OR "Вытеснение пива в буфер" OR "Ополаскивание после производства" OR ("Режим СIP вкл" AND "Мойка") OR "fb_Wash_In_DB".bWashPump1) AND NOT "mm1";
   IF "ww1" THEN "Косвенное окно1" := 100; END_IF;
   IF "cw1" THEN "Косвенное окно1" := 0; END_IF;
END_REGION

REGION Network 7: Насос бустерный M2
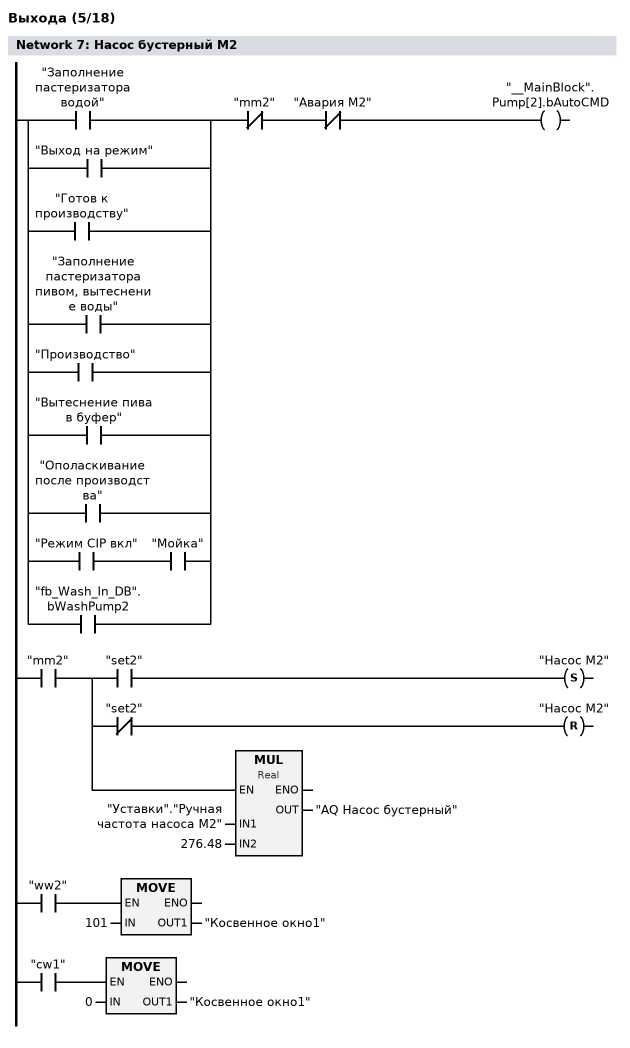
   RUNG wire#powerrail
      Contact( "Заполнение пастеризатора водой" )
      wire#w1
      I_Contact( "mm2" )
      I_Contact( "Авария М2" )
      Coil( "__MainBlock".Pump[2].bAutoCMD )
   END_RUNG
   RUNG wire#powerrail
      Contact( "Выход на режим" )
   END_RUNG wire#w1
   RUNG wire#powerrail
      Contact( "Готов к производству" )
   END_RUNG wire#w1
   RUNG wire#powerrail
      Contact( "Заполнение пастеризатора пивом, вытеснение воды" )
   END_RUNG wire#w1
   RUNG wire#powerrail
      Contact( "Производство" )
   END_RUNG wire#w1
   RUNG wire#powerrail
      Contact( "Вытеснение пива в буфер" )
   END_RUNG wire#w1
   RUNG wire#powerrail
      Contact( "Ополаскивание после производства" )
   END_RUNG wire#w1
   RUNG wire#powerrail
      Contact( "Режим СIP вкл" )
      Contact( "Мойка" )
   END_RUNG wire#w1
   RUNG wire#powerrail
      Contact( "fb_Wash_In_DB".bWashPump2 )
   END_RUNG wire#w1
   RUNG wire#powerrail
      Contact( "mm2" )
      wire#w2
      Contact( "set2" )
      S_Coil( "Насос М2" )
   END_RUNG
   RUNG wire#w2
      I_Contact( "set2" )
      R_Coil( "Насос М2" )
   END_RUNG
   RUNG wire#w2
      { S7_Templates := "SrcType := Real" } Mul(in1 := "Уставки"."Ручная частота насоса M2", in2 := 276.48, out => "AQ Насос бустерный")
   END_RUNG
   RUNG wire#powerrail
      Contact( "ww2" )
      Move(in := 101, out1 => "Косвенное окно1")
   END_RUNG
   RUNG wire#powerrail
      Contact( "cw1" )
      Move(in := 0, out1 => "Косвенное окно1")
   END_RUNG
   // the same network as SCL:
   "__MainBlock".Pump[2].bAutoCMD := ("Заполнение пастеризатора водой" OR "Выход на режим" OR "Готов к производству" OR "Заполнение пастеризатора пивом, вытеснение воды" OR "Производство" OR "Вытеснение пива в буфер" OR "Ополаскивание после производства" OR ("Режим СIP вкл" AND "Мойка") OR "fb_Wash_In_DB".bWashPump2) AND NOT "mm2" AND NOT "Авария М2";
   IF "mm2" AND "set2" THEN "Насос М2" := TRUE; END_IF;
   IF "mm2" AND NOT "set2" THEN "Насос М2" := FALSE; END_IF;
   IF "mm2" THEN "AQ Насос бустерный" := "Уставки"."Ручная частота насоса M2" * 276.48; END_IF;
   IF "ww2" THEN "Косвенное окно1" := 101; END_IF;
   IF "cw1" THEN "Косвенное окно1" := 0; END_IF;
END_REGION

REGION Network 8: Насос раздачи M3 (CIP-)
   // Убрал режим откачка была рядом с СИП вкл
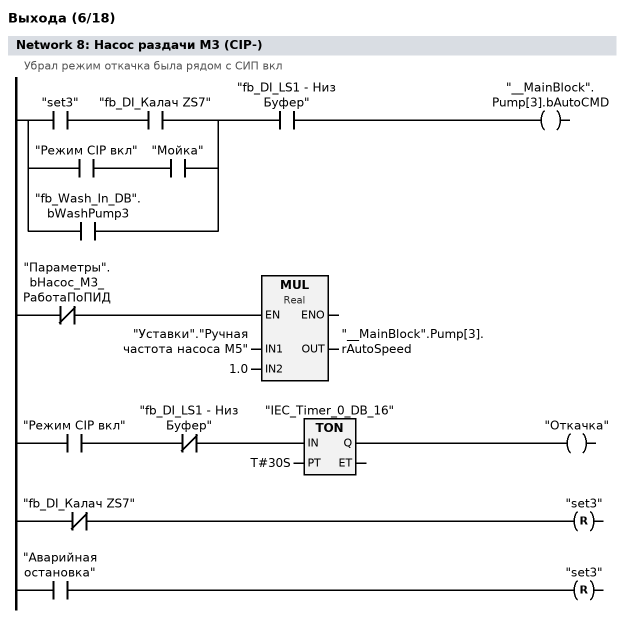
   "__MainBlock".Pump[3].bAutoCMD := (("set3" AND "fb_DI_Калач ZS7") OR ("Режим СIP вкл" AND "Мойка") OR "fb_Wash_In_DB".bWashPump3) AND "fb_DI_LS1 - Низ Буфер";
   IF NOT "Параметры".bНасос_М3_РаботаПоПИД THEN
       "__MainBlock".Pump[3].rAutoSpeed := "Уставки"."Ручная частота насоса M5" * 1.0;
   END_IF;
   "IEC_Timer_0_DB_16".TON(IN := "Режим СIP вкл" AND NOT "fb_DI_LS1 - Низ Буфер", PT := T#30S);
   "Откачка" := "IEC_Timer_0_DB_16".Q;
   IF NOT "fb_DI_Калач ZS7" THEN "set3" := FALSE; END_IF;
   IF "Аварийная остановка" THEN "set3" := FALSE; END_IF;
END_REGION

REGION Network 9: Насос ГВ пастеризации M-4
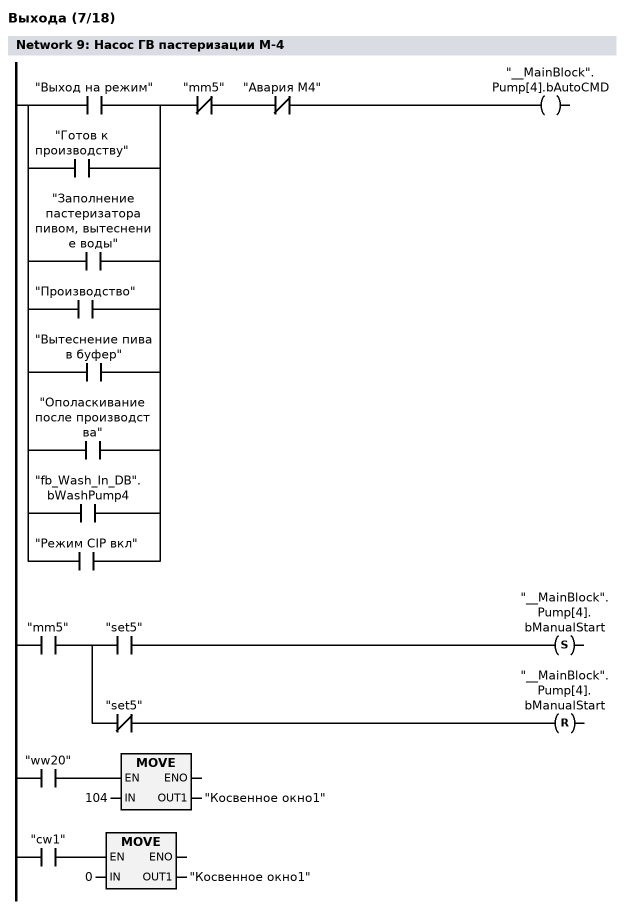
   RUNG wire#powerrail
      Contact( "Выход на режим" )
      wire#w1
      I_Contact( "mm5" )
      I_Contact( "Авария М4" )
      Coil( "__MainBlock".Pump[4].bAutoCMD )
   END_RUNG
   RUNG wire#powerrail
      Contact( "Готов к производству" )
   END_RUNG wire#w1
   RUNG wire#powerrail
      Contact( "Заполнение пастеризатора пивом, вытеснение воды" )
   END_RUNG wire#w1
   RUNG wire#powerrail
      Contact( "Производство" )
   END_RUNG wire#w1
   RUNG wire#powerrail
      Contact( "Вытеснение пива в буфер" )
   END_RUNG wire#w1
   RUNG wire#powerrail
      Contact( "Ополаскивание после производства" )
   END_RUNG wire#w1
   RUNG wire#powerrail
      Contact( "fb_Wash_In_DB".bWashPump4 )
   END_RUNG wire#w1
   RUNG wire#powerrail
      Contact( "Режим СIP вкл" )
   END_RUNG wire#w1
   RUNG wire#powerrail
      Contact( "mm5" )
      wire#w2
      Contact( "set5" )
      S_Coil( "__MainBlock".Pump[4].bManualStart )
   END_RUNG
   RUNG wire#w2
      I_Contact( "set5" )
      R_Coil( "__MainBlock".Pump[4].bManualStart )
   END_RUNG
   RUNG wire#powerrail
      Contact( "ww20" )
      Move(in := 104, out1 => "Косвенное окно1")
   END_RUNG
   RUNG wire#powerrail
      Contact( "cw1" )
      Move(in := 0, out1 => "Косвенное окно1")
   END_RUNG
   // the same network as SCL:
   "__MainBlock".Pump[4].bAutoCMD := ("Выход на режим" OR "Готов к производству" OR "Заполнение пастеризатора пивом, вытеснение воды" OR "Производство" OR "Вытеснение пива в буфер" OR "Ополаскивание после производства" OR "fb_Wash_In_DB".bWashPump4 OR "Режим СIP вкл") AND NOT "mm5" AND NOT "Авария М4";
   IF "mm5" AND "set5" THEN "__MainBlock".Pump[4].bManualStart := TRUE; END_IF;
   IF "mm5" AND NOT "set5" THEN "__MainBlock".Pump[4].bManualStart := FALSE; END_IF;
   IF "ww20" THEN "Косвенное окно1" := 104; END_IF;
   IF "cw1" THEN "Косвенное окно1" := 0; END_IF;
END_REGION

REGION Network 10: Насос секции охлаждения M-5
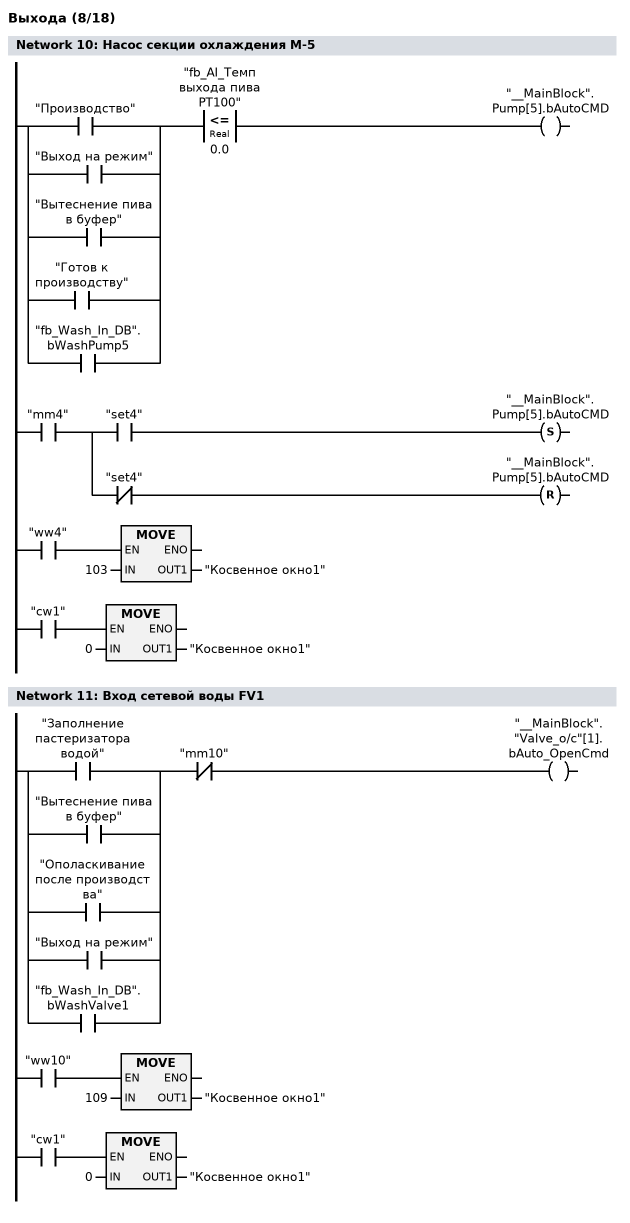
   RUNG wire#powerrail
      Contact( "Производство" )
      wire#w1
      { S7_Templates := "SrcType := Real" } LE_Contact(in1 := "fb_AI_Темп выхода пива  PT100", in2 := 0.0)
      Coil( "__MainBlock".Pump[5].bAutoCMD )
   END_RUNG
   RUNG wire#powerrail
      Contact( "Выход на режим" )
   END_RUNG wire#w1
   RUNG wire#powerrail
      Contact( "Вытеснение пива в буфер" )
   END_RUNG wire#w1
   RUNG wire#powerrail
      Contact( "Готов к производству" )
   END_RUNG wire#w1
   RUNG wire#powerrail
      Contact( "fb_Wash_In_DB".bWashPump5 )
   END_RUNG wire#w1
   RUNG wire#powerrail
      Contact( "mm4" )
      wire#w2
      Contact( "set4" )
      S_Coil( "__MainBlock".Pump[5].bAutoCMD )
   END_RUNG
   RUNG wire#w2
      I_Contact( "set4" )
      R_Coil( "__MainBlock".Pump[5].bAutoCMD )
   END_RUNG
   RUNG wire#powerrail
      Contact( "ww4" )
      Move(in := 103, out1 => "Косвенное окно1")
   END_RUNG
   RUNG wire#powerrail
      Contact( "cw1" )
      Move(in := 0, out1 => "Косвенное окно1")
   END_RUNG
   // the same network as SCL:
   "__MainBlock".Pump[5].bAutoCMD := ("Производство" OR "Выход на режим" OR "Вытеснение пива в буфер" OR "Готов к производству" OR "fb_Wash_In_DB".bWashPump5) AND ("fb_AI_Темп выхода пива  PT100" <= 0.0);
   IF "mm4" AND "set4" THEN "__MainBlock".Pump[5].bAutoCMD := TRUE; END_IF;
   IF "mm4" AND NOT "set4" THEN "__MainBlock".Pump[5].bAutoCMD := FALSE; END_IF;
   IF "ww4" THEN "Косвенное окно1" := 103; END_IF;
   IF "cw1" THEN "Косвенное окно1" := 0; END_IF;
END_REGION

REGION Network 11: Вход сетевой воды FV1
   RUNG wire#powerrail
      Contact( "Заполнение пастеризатора водой" )
      wire#w1
      I_Contact( "mm10" )
      Coil( "__MainBlock"."Valve_o/c"[1].bAuto_OpenCmd )
   END_RUNG
   RUNG wire#powerrail
      Contact( "Вытеснение пива в буфер" )
   END_RUNG wire#w1
   RUNG wire#powerrail
      Contact( "Ополаскивание после производства" )
   END_RUNG wire#w1
   RUNG wire#powerrail
      Contact( "Выход на режим" )
   END_RUNG wire#w1
   RUNG wire#powerrail
      Contact( "fb_Wash_In_DB".bWashValve1 )
   END_RUNG wire#w1
   RUNG wire#powerrail
      Contact( "ww10" )
      Move(in := 109, out1 => "Косвенное окно1")
   END_RUNG
   RUNG wire#powerrail
      Contact( "cw1" )
      Move(in := 0, out1 => "Косвенное окно1")
   END_RUNG
   // the same network as SCL:
   "__MainBlock"."Valve_o/c"[1].bAuto_OpenCmd := ("Заполнение пастеризатора водой" OR "Вытеснение пива в буфер" OR "Ополаскивание после производства" OR "Выход на режим" OR "fb_Wash_In_DB".bWashValve1) AND NOT "mm10";
   IF "ww10" THEN "Косвенное окно1" := 109; END_IF;
   IF "cw1" THEN "Косвенное окно1" := 0; END_IF;
END_REGION

REGION Network 12: Вход пива FV2
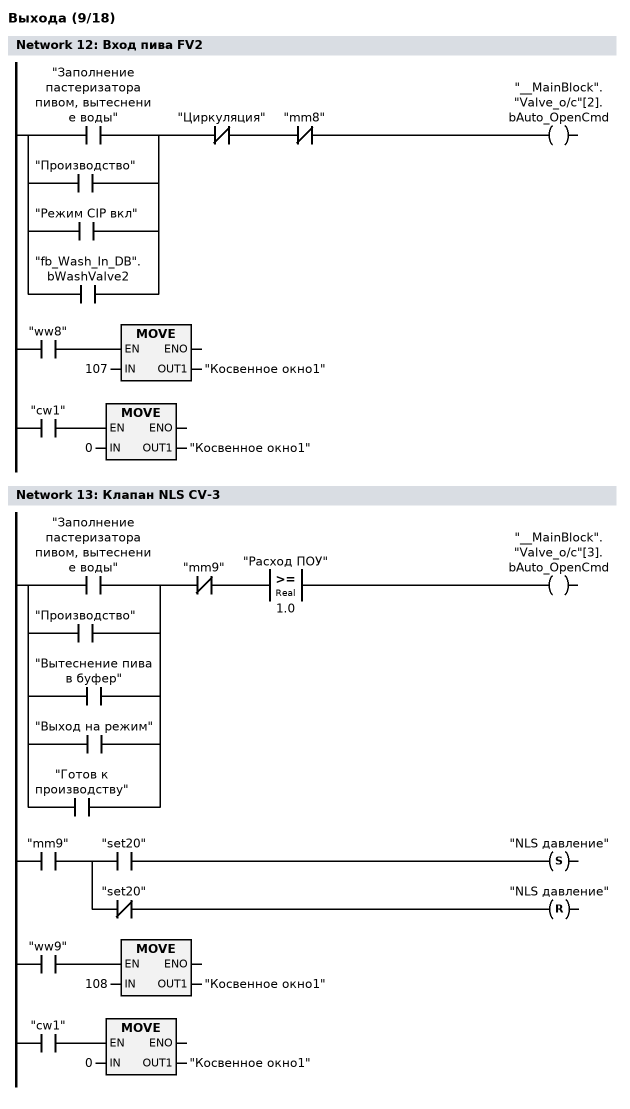
   RUNG wire#powerrail
      Contact( "Заполнение пастеризатора пивом, вытеснение воды" )
      wire#w1
      I_Contact( "Циркуляция" )
      I_Contact( "mm8" )
      Coil( "__MainBlock"."Valve_o/c"[2].bAuto_OpenCmd )
   END_RUNG
   RUNG wire#powerrail
      Contact( "Производство" )
   END_RUNG wire#w1
   RUNG wire#powerrail
      Contact( "Режим СIP вкл" )
   END_RUNG wire#w1
   RUNG wire#powerrail
      Contact( "fb_Wash_In_DB".bWashValve2 )
   END_RUNG wire#w1
   RUNG wire#powerrail
      Contact( "ww8" )
      Move(in := 107, out1 => "Косвенное окно1")
   END_RUNG
   RUNG wire#powerrail
      Contact( "cw1" )
      Move(in := 0, out1 => "Косвенное окно1")
   END_RUNG
   // the same network as SCL:
   "__MainBlock"."Valve_o/c"[2].bAuto_OpenCmd := ("Заполнение пастеризатора пивом, вытеснение воды" OR "Производство" OR "Режим СIP вкл" OR "fb_Wash_In_DB".bWashValve2) AND NOT "Циркуляция" AND NOT "mm8";
   IF "ww8" THEN "Косвенное окно1" := 107; END_IF;
   IF "cw1" THEN "Косвенное окно1" := 0; END_IF;
END_REGION

REGION Network 13: Клапан NLS CV-3
   RUNG wire#powerrail
      Contact( "Заполнение пастеризатора пивом, вытеснение воды" )
      wire#w1
      I_Contact( "mm9" )
      { S7_Templates := "SrcType := Real" } GE_Contact(in1 := "Расход ПОУ", in2 := 1.0)
      Coil( "__MainBlock"."Valve_o/c"[3].bAuto_OpenCmd )
   END_RUNG
   RUNG wire#powerrail
      Contact( "Производство" )
   END_RUNG wire#w1
   RUNG wire#powerrail
      Contact( "Вытеснение пива в буфер" )
   END_RUNG wire#w1
   RUNG wire#powerrail
      Contact( "Выход на режим" )
   END_RUNG wire#w1
   RUNG wire#powerrail
      Contact( "Готов к производству" )
   END_RUNG wire#w1
   RUNG wire#powerrail
      Contact( "mm9" )
      wire#w2
      Contact( "set20" )
      S_Coil( "NLS давление" )
   END_RUNG
   RUNG wire#w2
      I_Contact( "set20" )
      R_Coil( "NLS давление" )
   END_RUNG
   RUNG wire#powerrail
      Contact( "ww9" )
      Move(in := 108, out1 => "Косвенное окно1")
   END_RUNG
   RUNG wire#powerrail
      Contact( "cw1" )
      Move(in := 0, out1 => "Косвенное окно1")
   END_RUNG
   // the same network as SCL:
   "__MainBlock"."Valve_o/c"[3].bAuto_OpenCmd := ("Заполнение пастеризатора пивом, вытеснение воды" OR "Производство" OR "Вытеснение пива в буфер" OR "Выход на режим" OR "Готов к производству") AND NOT "mm9" AND ("Расход ПОУ" >= 1.0);
   IF "mm9" AND "set20" THEN "NLS давление" := TRUE; END_IF;
   IF "mm9" AND NOT "set20" THEN "NLS давление" := FALSE; END_IF;
   IF "ww9" THEN "Косвенное окно1" := 108; END_IF;
   IF "cw1" THEN "Косвенное окно1" := 0; END_IF;
END_REGION

REGION Network 14: Клапан циркуляции FV4
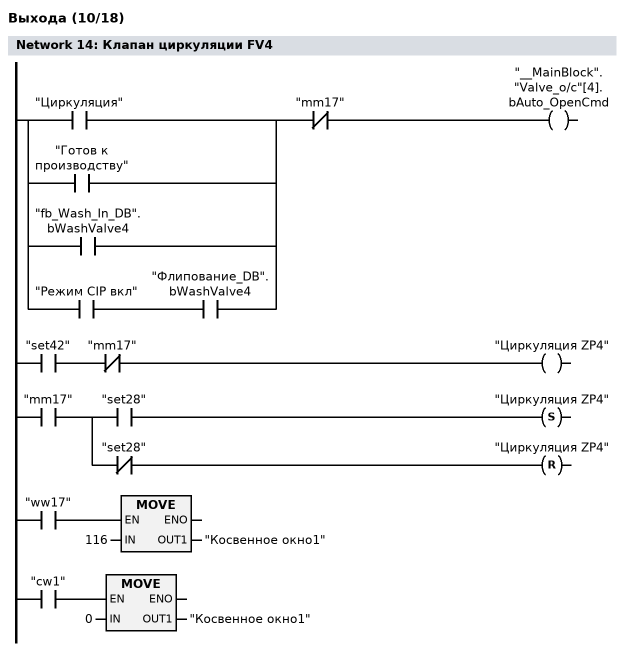
   RUNG wire#powerrail
      Contact( "Циркуляция" )
      wire#w1
      I_Contact( "mm17" )
      Coil( "__MainBlock"."Valve_o/c"[4].bAuto_OpenCmd )
   END_RUNG
   RUNG wire#powerrail
      Contact( "Готов к производству" )
   END_RUNG wire#w1
   RUNG wire#powerrail
      Contact( "fb_Wash_In_DB".bWashValve4 )
   END_RUNG wire#w1
   RUNG wire#powerrail
      Contact( "Режим СIP вкл" )
      Contact( "Флипование_DB".bWashValve4 )
   END_RUNG wire#w1
   RUNG wire#powerrail
      Contact( "set42" )
      I_Contact( "mm17" )
      Coil( "Циркуляция ZP4" )
   END_RUNG
   RUNG wire#powerrail
      Contact( "mm17" )
      wire#w2
      Contact( "set28" )
      S_Coil( "Циркуляция ZP4" )
   END_RUNG
   RUNG wire#w2
      I_Contact( "set28" )
      R_Coil( "Циркуляция ZP4" )
   END_RUNG
   RUNG wire#powerrail
      Contact( "ww17" )
      Move(in := 116, out1 => "Косвенное окно1")
   END_RUNG
   RUNG wire#powerrail
      Contact( "cw1" )
      Move(in := 0, out1 => "Косвенное окно1")
   END_RUNG
   // the same network as SCL:
   "__MainBlock"."Valve_o/c"[4].bAuto_OpenCmd := ("Циркуляция" OR "Готов к производству" OR "fb_Wash_In_DB".bWashValve4 OR ("Режим СIP вкл" AND "Флипование_DB".bWashValve4)) AND NOT "mm17";
   "Циркуляция ZP4" := "set42" AND NOT "mm17";
   IF "mm17" AND "set28" THEN "Циркуляция ZP4" := TRUE; END_IF;
   IF "mm17" AND NOT "set28" THEN "Циркуляция ZP4" := FALSE; END_IF;
   IF "ww17" THEN "Косвенное окно1" := 116; END_IF;
   IF "cw1" THEN "Косвенное окно1" := 0; END_IF;
END_REGION

REGION Network 15: Трап FV5
   // Клапан работает в инверсии
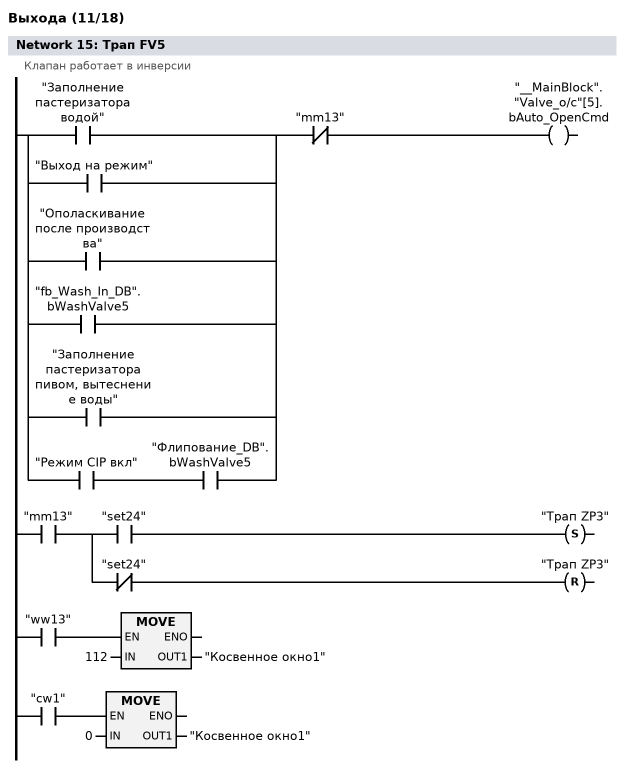
   RUNG wire#powerrail
      Contact( "Заполнение пастеризатора водой" )
      wire#w1
      I_Contact( "mm13" )
      Coil( "__MainBlock"."Valve_o/c"[5].bAuto_OpenCmd )
   END_RUNG
   RUNG wire#powerrail
      Contact( "Выход на режим" )
   END_RUNG wire#w1
   RUNG wire#powerrail
      Contact( "Ополаскивание после производства" )
   END_RUNG wire#w1
   RUNG wire#powerrail
      Contact( "fb_Wash_In_DB".bWashValve5 )
   END_RUNG wire#w1
   RUNG wire#powerrail
      Contact( "Заполнение пастеризатора пивом, вытеснение воды" )
   END_RUNG wire#w1
   RUNG wire#powerrail
      Contact( "Режим СIP вкл" )
      Contact( "Флипование_DB".bWashValve5 )
   END_RUNG wire#w1
   RUNG wire#powerrail
      Contact( "mm13" )
      wire#w2
      Contact( "set24" )
      S_Coil( "Трап ZP3" )
   END_RUNG
   RUNG wire#w2
      I_Contact( "set24" )
      R_Coil( "Трап ZP3" )
   END_RUNG
   RUNG wire#powerrail
      Contact( "ww13" )
      Move(in := 112, out1 => "Косвенное окно1")
   END_RUNG
   RUNG wire#powerrail
      Contact( "cw1" )
      Move(in := 0, out1 => "Косвенное окно1")
   END_RUNG
   // the same network as SCL:
   "__MainBlock"."Valve_o/c"[5].bAuto_OpenCmd := ("Заполнение пастеризатора водой" OR "Выход на режим" OR "Ополаскивание после производства" OR "fb_Wash_In_DB".bWashValve5 OR "Заполнение пастеризатора пивом, вытеснение воды" OR ("Режим СIP вкл" AND "Флипование_DB".bWashValve5)) AND NOT "mm13";
   IF "mm13" AND "set24" THEN "Трап ZP3" := TRUE; END_IF;
   IF "mm13" AND NOT "set24" THEN "Трап ZP3" := FALSE; END_IF;
   IF "ww13" THEN "Косвенное окно1" := 112; END_IF;
   IF "cw1" THEN "Косвенное окно1" := 0; END_IF;
END_REGION

REGION Network 16: Клапан Возврата FV6
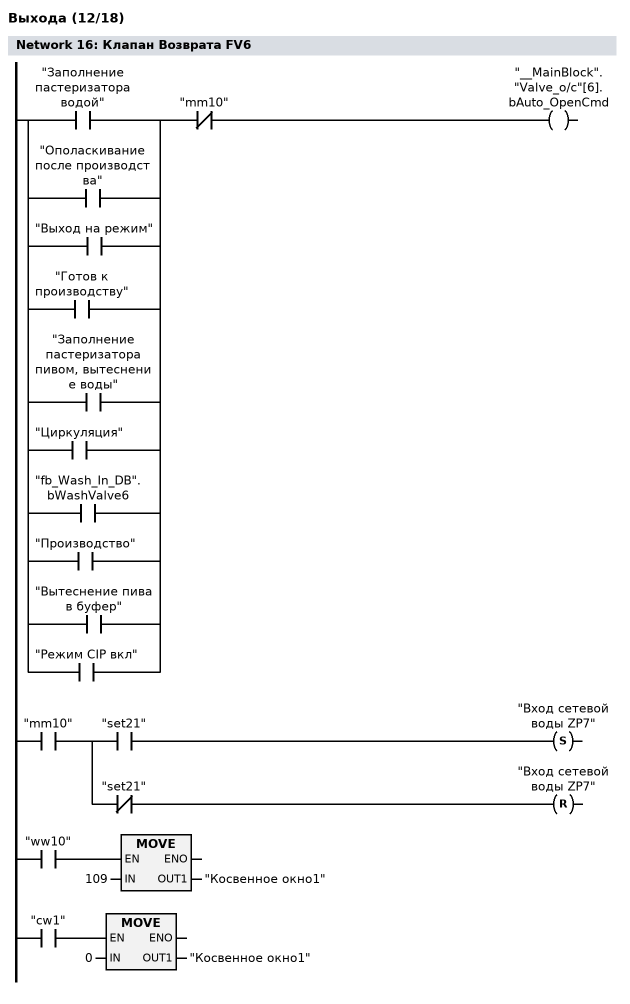
   RUNG wire#powerrail
      Contact( "Заполнение пастеризатора водой" )
      wire#w1
      I_Contact( "mm10" )
      Coil( "__MainBlock"."Valve_o/c"[6].bAuto_OpenCmd )
   END_RUNG
   RUNG wire#powerrail
      Contact( "Ополаскивание после производства" )
   END_RUNG wire#w1
   RUNG wire#powerrail
      Contact( "Выход на режим" )
   END_RUNG wire#w1
   RUNG wire#powerrail
      Contact( "Готов к производству" )
   END_RUNG wire#w1
   RUNG wire#powerrail
      Contact( "Заполнение пастеризатора пивом, вытеснение воды" )
   END_RUNG wire#w1
   RUNG wire#powerrail
      Contact( "Циркуляция" )
   END_RUNG wire#w1
   RUNG wire#powerrail
      Contact( "fb_Wash_In_DB".bWashValve6 )
   END_RUNG wire#w1
   RUNG wire#powerrail
      Contact( "Производство" )
   END_RUNG wire#w1
   RUNG wire#powerrail
      Contact( "Вытеснение пива в буфер" )
   END_RUNG wire#w1
   RUNG wire#powerrail
      Contact( "Режим СIP вкл" )
   END_RUNG wire#w1
   RUNG wire#powerrail
      Contact( "mm10" )
      wire#w2
      Contact( "set21" )
      S_Coil( "Вход сетевой воды ZP7" )
   END_RUNG
   RUNG wire#w2
      I_Contact( "set21" )
      R_Coil( "Вход сетевой воды ZP7" )
   END_RUNG
   RUNG wire#powerrail
      Contact( "ww10" )
      Move(in := 109, out1 => "Косвенное окно1")
   END_RUNG
   RUNG wire#powerrail
      Contact( "cw1" )
      Move(in := 0, out1 => "Косвенное окно1")
   END_RUNG
   // the same network as SCL:
   "__MainBlock"."Valve_o/c"[6].bAuto_OpenCmd := ("Заполнение пастеризатора водой" OR "Ополаскивание после производства" OR "Выход на режим" OR "Готов к производству" OR "Заполнение пастеризатора пивом, вытеснение воды" OR "Циркуляция" OR "fb_Wash_In_DB".bWashValve6 OR "Производство" OR "Вытеснение пива в буфер" OR "Режим СIP вкл") AND NOT "mm10";
   IF "mm10" AND "set21" THEN "Вход сетевой воды ZP7" := TRUE; END_IF;
   IF "mm10" AND NOT "set21" THEN "Вход сетевой воды ZP7" := FALSE; END_IF;
   IF "ww10" THEN "Косвенное окно1" := 109; END_IF;
   IF "cw1" THEN "Косвенное окно1" := 0; END_IF;
END_REGION

REGION Network 17: Моющая Головка буфер FV7
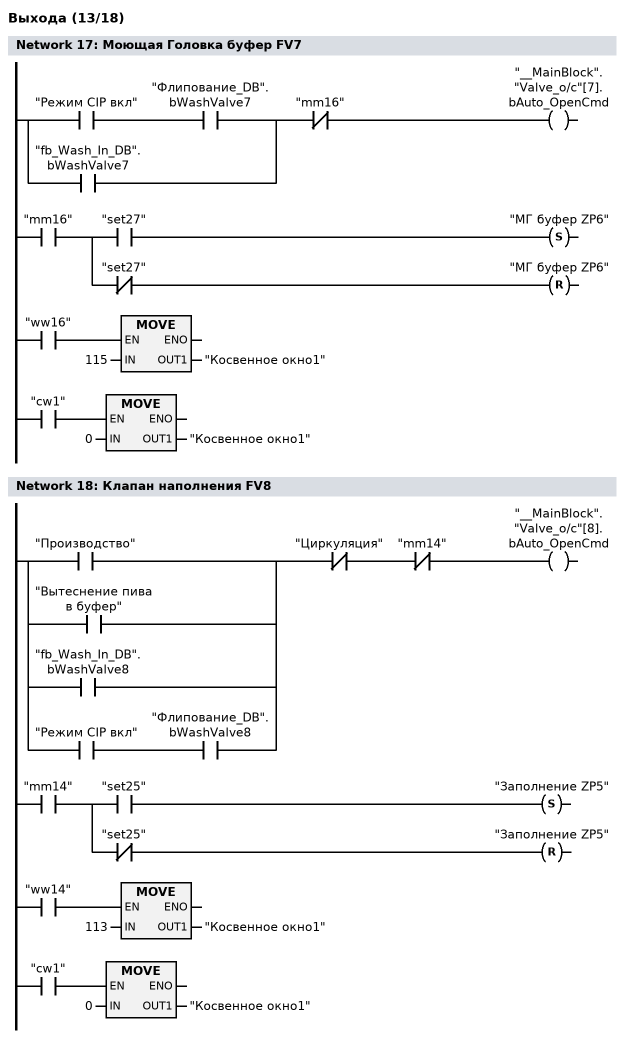
   RUNG wire#powerrail
      Contact( "Режим СIP вкл" )
      Contact( "Флипование_DB".bWashValve7 )
      wire#w1
      I_Contact( "mm16" )
      Coil( "__MainBlock"."Valve_o/c"[7].bAuto_OpenCmd )
   END_RUNG
   RUNG wire#powerrail
      Contact( "fb_Wash_In_DB".bWashValve7 )
   END_RUNG wire#w1
   RUNG wire#powerrail
      Contact( "mm16" )
      wire#w2
      Contact( "set27" )
      S_Coil( "МГ буфер ZP6" )
   END_RUNG
   RUNG wire#w2
      I_Contact( "set27" )
      R_Coil( "МГ буфер ZP6" )
   END_RUNG
   RUNG wire#powerrail
      Contact( "ww16" )
      Move(in := 115, out1 => "Косвенное окно1")
   END_RUNG
   RUNG wire#powerrail
      Contact( "cw1" )
      Move(in := 0, out1 => "Косвенное окно1")
   END_RUNG
   // the same network as SCL:
   "__MainBlock"."Valve_o/c"[7].bAuto_OpenCmd := (("Режим СIP вкл" AND "Флипование_DB".bWashValve7) OR "fb_Wash_In_DB".bWashValve7) AND NOT "mm16";
   IF "mm16" AND "set27" THEN "МГ буфер ZP6" := TRUE; END_IF;
   IF "mm16" AND NOT "set27" THEN "МГ буфер ZP6" := FALSE; END_IF;
   IF "ww16" THEN "Косвенное окно1" := 115; END_IF;
   IF "cw1" THEN "Косвенное окно1" := 0; END_IF;
END_REGION

REGION Network 18: Клапан наполнения FV8
   RUNG wire#powerrail
      Contact( "Производство" )
      wire#w1
      I_Contact( "Циркуляция" )
      I_Contact( "mm14" )
      Coil( "__MainBlock"."Valve_o/c"[8].bAuto_OpenCmd )
   END_RUNG
   RUNG wire#powerrail
      Contact( "Вытеснение пива в буфер" )
   END_RUNG wire#w1
   RUNG wire#powerrail
      Contact( "fb_Wash_In_DB".bWashValve8 )
   END_RUNG wire#w1
   RUNG wire#powerrail
      Contact( "Режим СIP вкл" )
      Contact( "Флипование_DB".bWashValve8 )
   END_RUNG wire#w1
   RUNG wire#powerrail
      Contact( "mm14" )
      wire#w2
      Contact( "set25" )
      S_Coil( "Заполнение ZP5" )
   END_RUNG
   RUNG wire#w2
      I_Contact( "set25" )
      R_Coil( "Заполнение ZP5" )
   END_RUNG
   RUNG wire#powerrail
      Contact( "ww14" )
      Move(in := 113, out1 => "Косвенное окно1")
   END_RUNG
   RUNG wire#powerrail
      Contact( "cw1" )
      Move(in := 0, out1 => "Косвенное окно1")
   END_RUNG
   // the same network as SCL:
   "__MainBlock"."Valve_o/c"[8].bAuto_OpenCmd := ("Производство" OR "Вытеснение пива в буфер" OR "fb_Wash_In_DB".bWashValve8 OR ("Режим СIP вкл" AND "Флипование_DB".bWashValve8)) AND NOT "Циркуляция" AND NOT "mm14";
   IF "mm14" AND "set25" THEN "Заполнение ZP5" := TRUE; END_IF;
   IF "mm14" AND NOT "set25" THEN "Заполнение ZP5" := FALSE; END_IF;
   IF "ww14" THEN "Косвенное окно1" := 113; END_IF;
   IF "cw1" THEN "Косвенное окно1" := 0; END_IF;
END_REGION

REGION Network 19: Клапан розлива FV9
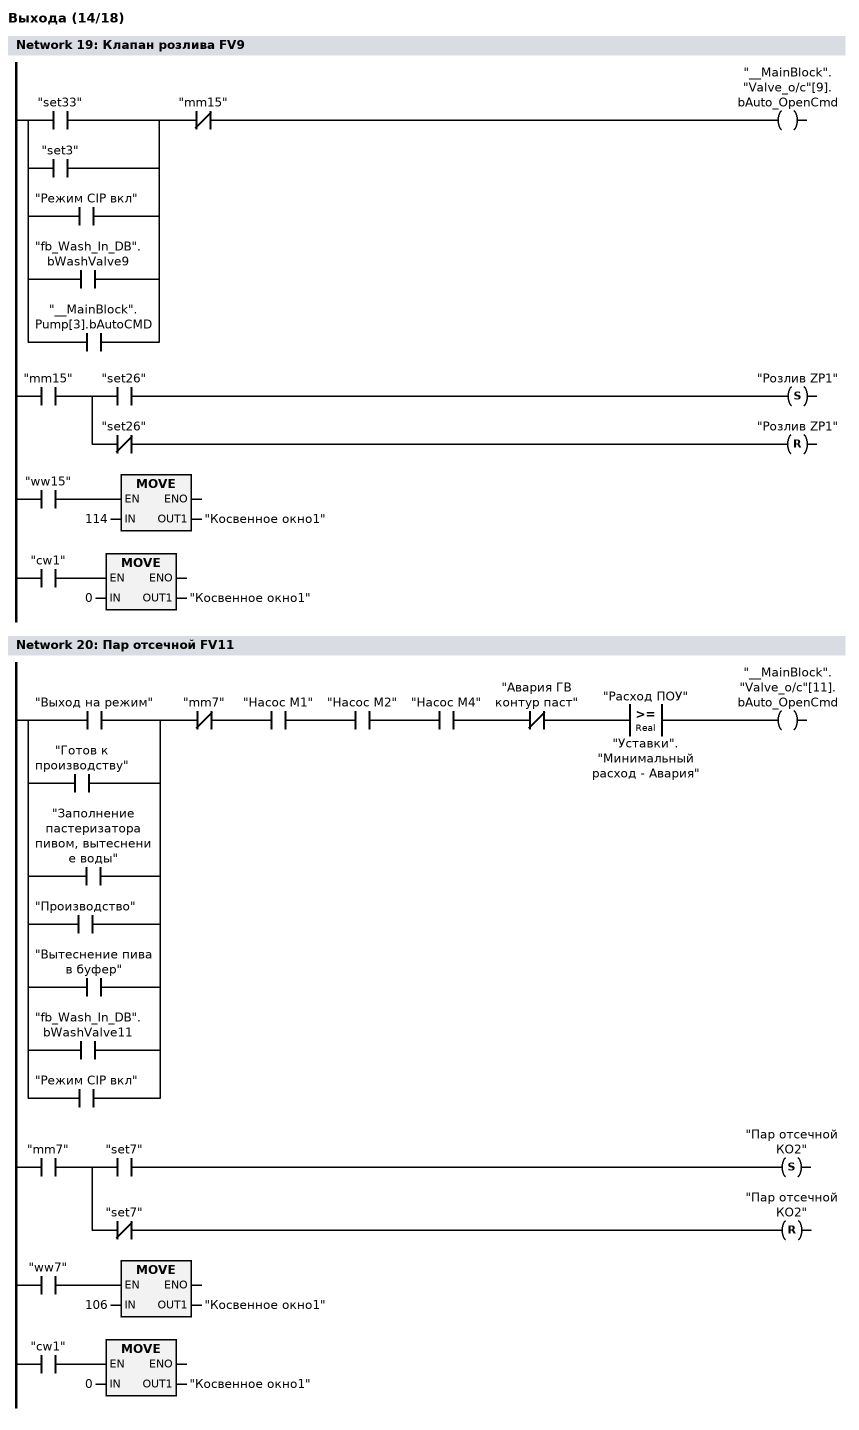
   RUNG wire#powerrail
      Contact( "set33" )
      wire#w1
      I_Contact( "mm15" )
      Coil( "__MainBlock"."Valve_o/c"[9].bAuto_OpenCmd )
   END_RUNG
   RUNG wire#powerrail
      Contact( "set3" )
   END_RUNG wire#w1
   RUNG wire#powerrail
      Contact( "Режим СIP вкл" )
   END_RUNG wire#w1
   RUNG wire#powerrail
      Contact( "fb_Wash_In_DB".bWashValve9 )
   END_RUNG wire#w1
   RUNG wire#powerrail
      Contact( "__MainBlock".Pump[3].bAutoCMD )
   END_RUNG wire#w1
   RUNG wire#powerrail
      Contact( "mm15" )
      wire#w2
      Contact( "set26" )
      S_Coil( "Розлив ZP1" )
   END_RUNG
   RUNG wire#w2
      I_Contact( "set26" )
      R_Coil( "Розлив ZP1" )
   END_RUNG
   RUNG wire#powerrail
      Contact( "ww15" )
      Move(in := 114, out1 => "Косвенное окно1")
   END_RUNG
   RUNG wire#powerrail
      Contact( "cw1" )
      Move(in := 0, out1 => "Косвенное окно1")
   END_RUNG
   // the same network as SCL:
   "__MainBlock"."Valve_o/c"[9].bAuto_OpenCmd := ("set33" OR "set3" OR "Режим СIP вкл" OR "fb_Wash_In_DB".bWashValve9 OR "__MainBlock".Pump[3].bAutoCMD) AND NOT "mm15";
   IF "mm15" AND "set26" THEN "Розлив ZP1" := TRUE; END_IF;
   IF "mm15" AND NOT "set26" THEN "Розлив ZP1" := FALSE; END_IF;
   IF "ww15" THEN "Косвенное окно1" := 114; END_IF;
   IF "cw1" THEN "Косвенное окно1" := 0; END_IF;
END_REGION

REGION Network 20: Пар отсечной FV11
   RUNG wire#powerrail
      Contact( "Выход на режим" )
      wire#w1
      I_Contact( "mm7" )
      Contact( "Насос М1" )
      Contact( "Насос М2" )
      Contact( "Насос М4" )
      I_Contact( "Авария ГВ контур паст" )
      { S7_Templates := "SrcType := Real" } GE_Contact(in1 := "Расход ПОУ", in2 := "Уставки"."Минимальный расход - Авария")
      Coil( "__MainBlock"."Valve_o/c"[11].bAuto_OpenCmd )
   END_RUNG
   RUNG wire#powerrail
      Contact( "Готов к производству" )
   END_RUNG wire#w1
   RUNG wire#powerrail
      Contact( "Заполнение пастеризатора пивом, вытеснение воды" )
   END_RUNG wire#w1
   RUNG wire#powerrail
      Contact( "Производство" )
   END_RUNG wire#w1
   RUNG wire#powerrail
      Contact( "Вытеснение пива в буфер" )
   END_RUNG wire#w1
   RUNG wire#powerrail
      Contact( "fb_Wash_In_DB".bWashValve11 )
   END_RUNG wire#w1
   RUNG wire#powerrail
      Contact( "Режим СIP вкл" )
   END_RUNG wire#w1
   RUNG wire#powerrail
      Contact( "mm7" )
      wire#w2
      Contact( "set7" )
      S_Coil( "Пар отсечной КО2" )
   END_RUNG
   RUNG wire#w2
      I_Contact( "set7" )
      R_Coil( "Пар отсечной КО2" )
   END_RUNG
   RUNG wire#powerrail
      Contact( "ww7" )
      Move(in := 106, out1 => "Косвенное окно1")
   END_RUNG
   RUNG wire#powerrail
      Contact( "cw1" )
      Move(in := 0, out1 => "Косвенное окно1")
   END_RUNG
   // the same network as SCL:
   "__MainBlock"."Valve_o/c"[11].bAuto_OpenCmd := ("Выход на режим" OR "Готов к производству" OR "Заполнение пастеризатора пивом, вытеснение воды" OR "Производство" OR "Вытеснение пива в буфер" OR "fb_Wash_In_DB".bWashValve11 OR "Режим СIP вкл") AND NOT "mm7" AND "Насос М1" AND "Насос М2" AND "Насос М4" AND NOT "Авария ГВ контур паст" AND ("Расход ПОУ" >= "Уставки"."Минимальный расход - Авария");
   IF "mm7" AND "set7" THEN "Пар отсечной КО2" := TRUE; END_IF;
   IF "mm7" AND NOT "set7" THEN "Пар отсечной КО2" := FALSE; END_IF;
   IF "ww7" THEN "Косвенное окно1" := 106; END_IF;
   IF "cw1" THEN "Косвенное окно1" := 0; END_IF;
END_REGION

REGION Network 21: Вход пропиленгликоль FV12
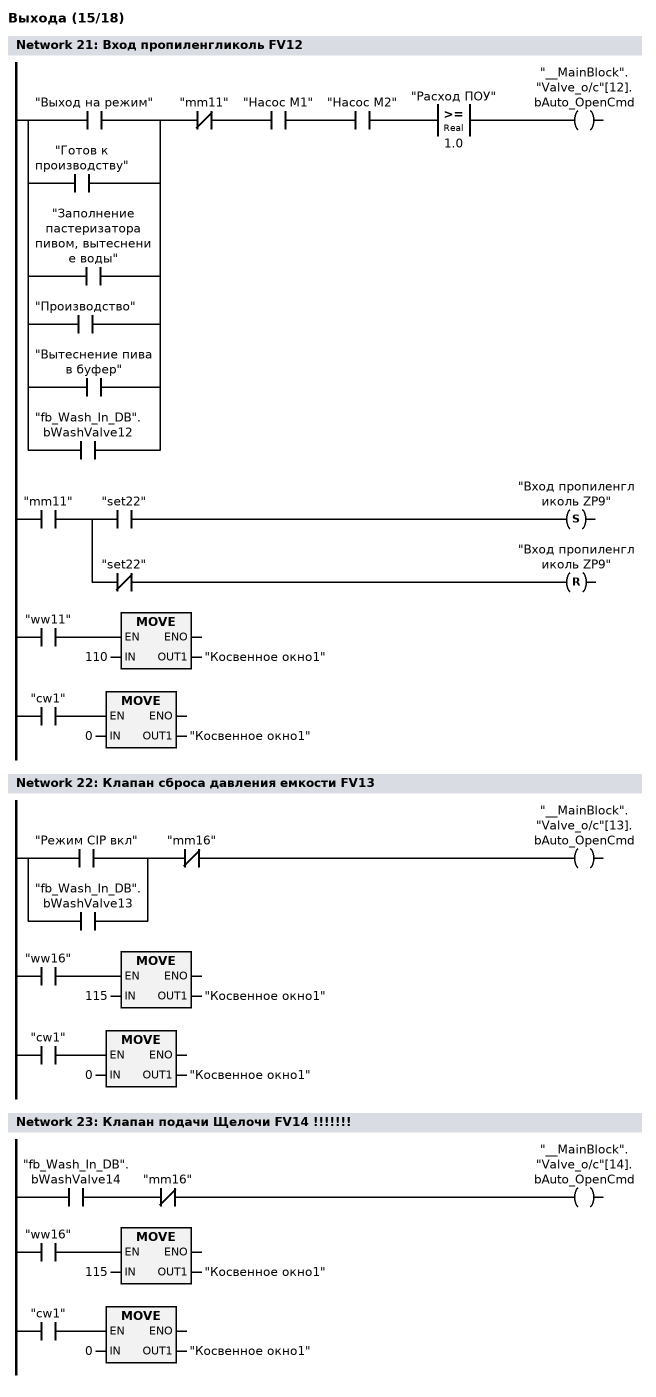
   RUNG wire#powerrail
      Contact( "Выход на режим" )
      wire#w1
      I_Contact( "mm11" )
      Contact( "Насос М1" )
      Contact( "Насос М2" )
      { S7_Templates := "SrcType := Real" } GE_Contact(in1 := "Расход ПОУ", in2 := 1.0)
      Coil( "__MainBlock"."Valve_o/c"[12].bAuto_OpenCmd )
   END_RUNG
   RUNG wire#powerrail
      Contact( "Готов к производству" )
   END_RUNG wire#w1
   RUNG wire#powerrail
      Contact( "Заполнение пастеризатора пивом, вытеснение воды" )
   END_RUNG wire#w1
   RUNG wire#powerrail
      Contact( "Производство" )
   END_RUNG wire#w1
   RUNG wire#powerrail
      Contact( "Вытеснение пива в буфер" )
   END_RUNG wire#w1
   RUNG wire#powerrail
      Contact( "fb_Wash_In_DB".bWashValve12 )
   END_RUNG wire#w1
   RUNG wire#powerrail
      Contact( "mm11" )
      wire#w2
      Contact( "set22" )
      S_Coil( "Вход пропиленгликоль ZP9" )
   END_RUNG
   RUNG wire#w2
      I_Contact( "set22" )
      R_Coil( "Вход пропиленгликоль ZP9" )
   END_RUNG
   RUNG wire#powerrail
      Contact( "ww11" )
      Move(in := 110, out1 => "Косвенное окно1")
   END_RUNG
   RUNG wire#powerrail
      Contact( "cw1" )
      Move(in := 0, out1 => "Косвенное окно1")
   END_RUNG
   // the same network as SCL:
   "__MainBlock"."Valve_o/c"[12].bAuto_OpenCmd := ("Выход на режим" OR "Готов к производству" OR "Заполнение пастеризатора пивом, вытеснение воды" OR "Производство" OR "Вытеснение пива в буфер" OR "fb_Wash_In_DB".bWashValve12) AND NOT "mm11" AND "Насос М1" AND "Насос М2" AND ("Расход ПОУ" >= 1.0);
   IF "mm11" AND "set22" THEN "Вход пропиленгликоль ZP9" := TRUE; END_IF;
   IF "mm11" AND NOT "set22" THEN "Вход пропиленгликоль ZP9" := FALSE; END_IF;
   IF "ww11" THEN "Косвенное окно1" := 110; END_IF;
   IF "cw1" THEN "Косвенное окно1" := 0; END_IF;
END_REGION

REGION Network 22: Клапан сброса давления емкости FV13
   RUNG wire#powerrail
      Contact( "Режим СIP вкл" )
      wire#w1
      I_Contact( "mm16" )
      Coil( "__MainBlock"."Valve_o/c"[13].bAuto_OpenCmd )
   END_RUNG
   RUNG wire#powerrail
      Contact( "fb_Wash_In_DB".bWashValve13 )
   END_RUNG wire#w1
   RUNG wire#powerrail
      Contact( "ww16" )
      Move(in := 115, out1 => "Косвенное окно1")
   END_RUNG
   RUNG wire#powerrail
      Contact( "cw1" )
      Move(in := 0, out1 => "Косвенное окно1")
   END_RUNG
   // the same network as SCL:
   "__MainBlock"."Valve_o/c"[13].bAuto_OpenCmd := ("Режим СIP вкл" OR "fb_Wash_In_DB".bWashValve13) AND NOT "mm16";
   IF "ww16" THEN "Косвенное окно1" := 115; END_IF;
   IF "cw1" THEN "Косвенное окно1" := 0; END_IF;
END_REGION

REGION Network 23: Клапан подачи Щелочи FV14 !!!!!!!
   RUNG wire#powerrail
      Contact( "fb_Wash_In_DB".bWashValve14 )
      I_Contact( "mm16" )
      Coil( "__MainBlock"."Valve_o/c"[14].bAuto_OpenCmd )
   END_RUNG
   RUNG wire#powerrail
      Contact( "ww16" )
      Move(in := 115, out1 => "Косвенное окно1")
   END_RUNG
   RUNG wire#powerrail
      Contact( "cw1" )
      Move(in := 0, out1 => "Косвенное окно1")
   END_RUNG
   // the same network as SCL:
   "__MainBlock"."Valve_o/c"[14].bAuto_OpenCmd := "fb_Wash_In_DB".bWashValve14 AND NOT "mm16";
   IF "ww16" THEN "Косвенное окно1" := 115; END_IF;
   IF "cw1" THEN "Косвенное окно1" := 0; END_IF;
END_REGION

REGION Network 24: Насос щелочи
